FUNCTION "Indication" : Void   // FC11, SCL
{ S7_Optimized_Access := 'TRUE' }
VERSION : 0.1
BEGIN
   (*Управление индикацией*)
   //генератор импульсов
   "Timer_IND_1_DB".TON(IN := "Timer".IND_1_IN,
                        PT := "Timer".IND_1_PT,
                        Q => "Timer".IND_1_Q);
   "Timer_IND_2_DB".TON(IN := "Timer".IND_2_IN,
                        PT := "Timer".IND_2_PT,
                        Q => "Timer".IND_2_Q);
   "Timer".IND_1_PT := T#1s;
   "Timer".IND_2_PT := T#1s;
   IF NOT "Timer".IND_1_IN AND NOT "Timer".IND_2_IN THEN
       "Timer".IND_1_IN := TRUE;
   END_IF;
   IF "Timer".IND_1_Q THEN
       "Timer".IND_1_IN := FALSE;
       "Timer".IND_2_IN := TRUE;
       "Gen_imp" := FALSE;
   END_IF;
   IF "Timer".IND_2_Q THEN
       "Timer".IND_2_IN := FALSE;
       "Timer".IND_1_IN := TRUE;
       "Gen_imp" := TRUE;
   END_IF;

   (*Индикация «Работа»*)
   IF "Technology".Regim <> 5 AND
       "Technology".Regim <> 6 AND
       "Technology".Regim <> 7 AND
       "Technology".Regim <> 8 THEN
       "Sensors".Indication_RUN.Value := FALSE;
   END_IF;
   IF "Technology".Regim = 5 OR
       "Technology".Regim = 6 OR
       "Technology".Regim = 7 THEN
       "Sensors".Indication_RUN.Value := "Gen_imp";
   END_IF;
   IF "Technology".Regim = 8 THEN
       "Sensors".Indication_RUN.Value := TRUE;
   END_IF;

   (*Индикация «Авария»*)
   IF "Alarms_and_warnings".Alarm_P_gas_before_BG_max OR
       "Alarms_and_warnings".Alarm_P_gas_before_BG_min OR
       "Alarms_and_warnings".Alarm_P_gas_before_burner_min OR
       "Alarms_and_warnings".Alarm_P_gas_before_burner_max OR
       "Alarms_and_warnings".Alarm_DS_off OR
       "Alarms_and_warnings".Alarm_DV_off OR
       "Alarms_and_warnings".Alarm_dP_furnace_boiler_min OR
       "Alarms_and_warnings".Alarm_P_air_before_burner_min OR
       "Alarms_and_warnings".Alarm_P_water_after_boiler_min OR
       "Alarms_and_warnings".Alarm_P_water_after_boiler_max OR
       "Alarms_and_warnings".Alarm_T_water_after_boiler_max OR
       "Alarms_and_warnings".Alarm_Q_water_boiler_min OR
       "Alarms_and_warnings".Alarm_Not_flame_burner OR
       "Alarms_and_warnings".Alarm_stop_HMI OR
       "Alarms_and_warnings".Alarm_stop_SCADA OR
       "Alarms_and_warnings".Alarm_CO2_porog2 OR
       "Alarms_and_warnings".Alarm_CH4 THEN
       "Sensors".Indication_ALARM.Value := TRUE;
   ELSE
       IF "TON_alarm_1_DB".IN OR
           "TON_alarm_2_DB".IN OR
           "TON_alarm_3_DB".IN OR
           "TON_alarm_4_DB".IN OR
           "TON_alarm_5_DB".IN OR
           "TON_alarm_6_DB".IN OR
           "TON_alarm_7_DB".IN OR
           "TON_alarm_8_DB".IN OR
           "TON_alarm_9_DB".IN OR
           "TON_alarm_10_DB".IN OR
           "TON_alarm_11_DB".IN OR
           "TON_alarm_12_DB".IN OR
           "TON_alarm_13_DB".IN OR
           "FRONT_Btn_Alarm_stop_HMI" OR
           "FRONT_Btn_Alarm_stop_SCADA" OR
           "TON_alarm_14_DB".IN OR
           "TON_alarm_15_DB".IN THEN
           "Sensors".Indication_ALARM.Value := "Gen_imp";
       ELSE
           "Sensors".Indication_ALARM.Value := FALSE;
       END_IF;
   END_IF;

   (*Индикация «Защиты в норме»*)
   IF "Protections".Global THEN
       "Sensors".Indication_NORMA.Value := FALSE;
   ELSE
       IF "Protections".BLOCK_P_gas_before_BG_max OR
           "Protections".BLOCK_P_gas_before_BG_min OR
           "Protections".BLOCK_P_gas_before_burner_min OR
           "Protections".BLOCK_P_gas_before_burner_max OR
           "Protections".BLOCK_DS_off OR
           "Protections".BLOCK_DV_off OR
           "Protections".BLOCK_dP_in_furnance_min OR
           "Protections".BLOCK_P_air_before_burner_min OR
           "Protections".BLOCK_P_water_after_boiler_min OR
           "Protections".BLOCK_P_water_after_boiler_max OR
           "Protections".BLOCK_T_water_after_boiler_max OR
           "Protections".BLOCK_Q_water_boiler_min OR
           "Protections".BLOCK_Not_flame_burner OR
           "Protections".BLOCK_Alarm_stop_HMI OR
           "Protections".BLOCK_Alarm_stop_SCADA OR
           "Protections".BLOCK_CO2_porog2 OR
           "Protections".BLOCK_CH4 THEN
           "Sensors".Indication_NORMA.Value := "Gen_imp";
       ELSE
           "Sensors".Indication_NORMA.Value := TRUE;
       END_IF;
   END_IF;

   (*Индикация «Готов к розжигу»*)
   IF "Technology".Regim = 3 AND "Technology".Regim_ventilation_step = 25 THEN
       "Sensors".Indication_READY.Value := "Gen_imp";
   ELSE
       "Sensors".Indication_READY.Value := FALSE;
   END_IF;
END_FUNCTION

FUNCTION "Regim_map" : Void   // FC24, SCL
{ S7_Optimized_Access := 'TRUE' }
VERSION : 0.1
BEGIN
   (*Защита от неправильного ввода параметров режимной карты*)
   IF "RegMap".P_gaz_2 < "RegMap".P_gaz_1 THEN
       "RegMap".P_gaz_2 := "RegMap".P_gaz_1;
   END_IF;
   IF "RegMap".P_gaz_3 < "RegMap".P_gaz_2 THEN
       "RegMap".P_gaz_3 := "RegMap".P_gaz_2;
   END_IF;
   IF "RegMap".P_gaz_4 < "RegMap".P_gaz_3 THEN
       "RegMap".P_gaz_4 := "RegMap".P_gaz_3;
   END_IF;
   IF "RegMap".P_gaz_5 < "RegMap".P_gaz_4 THEN
       "RegMap".P_gaz_5 := "RegMap".P_gaz_4;
   END_IF;
   IF "RegMap".P_gaz_6 < "RegMap".P_gaz_5 THEN
       "RegMap".P_gaz_6 := "RegMap".P_gaz_5;
   END_IF;
   IF "RegMap".P_gaz_7 < "RegMap".P_gaz_6 THEN
       "RegMap".P_gaz_7 := "RegMap".P_gaz_6;
   END_IF;
   IF "RegMap".P_gaz_8 < "RegMap".P_gaz_7 THEN
       "RegMap".P_gaz_8 := "RegMap".P_gaz_7;
   END_IF;

   (*НАСТРОЙКА РЕЖИМНОЙ КАРТЫ*)
   (*давление воздуха*)
   "Polyline_P_air_DB"();

   "Polyline_P_air_DB".Input := "Sensors".P_gas_before_burner.Value;

   "Polyline_P_air_DB".UserData.Point[1].x := "RegMap".P_gaz_1;
   "Polyline_P_air_DB".UserData.Point[2].x := "RegMap".P_gaz_2;
   "Polyline_P_air_DB".UserData.Point[3].x := "RegMap".P_gaz_3;
   "Polyline_P_air_DB".UserData.Point[4].x := "RegMap".P_gaz_4;
   "Polyline_P_air_DB".UserData.Point[5].x := "RegMap".P_gaz_5;
   "Polyline_P_air_DB".UserData.Point[6].x := "RegMap".P_gaz_6;
   "Polyline_P_air_DB".UserData.Point[7].x := "RegMap".P_gaz_7;
   "Polyline_P_air_DB".UserData.Point[8].x := "RegMap".P_gaz_8;

   "Polyline_P_air_DB".UserData.Point[1].y := "RegMap".P_air_1;
   "Polyline_P_air_DB".UserData.Point[2].y := "RegMap".P_air_2;
   "Polyline_P_air_DB".UserData.Point[3].y := "RegMap".P_air_3;
   "Polyline_P_air_DB".UserData.Point[4].y := "RegMap".P_air_4;
   "Polyline_P_air_DB".UserData.Point[5].y := "RegMap".P_air_5;
   "Polyline_P_air_DB".UserData.Point[6].y := "RegMap".P_air_6;
   "Polyline_P_air_DB".UserData.Point[7].y := "RegMap".P_air_7;
   "Polyline_P_air_DB".UserData.Point[8].y := "RegMap".P_air_8;

   (*разряжение*)
   "Polyline_dP_DB"();

   "Polyline_dP_DB".Input := "Sensors".P_gas_before_burner.Value;

   "Polyline_dP_DB".UserData.Point[1].x := "RegMap".P_gaz_1;
   "Polyline_dP_DB".UserData.Point[2].x := "RegMap".P_gaz_2;
   "Polyline_dP_DB".UserData.Point[3].x := "RegMap".P_gaz_3;
   "Polyline_dP_DB".UserData.Point[4].x := "RegMap".P_gaz_4;
   "Polyline_dP_DB".UserData.Point[5].x := "RegMap".P_gaz_5;
   "Polyline_dP_DB".UserData.Point[6].x := "RegMap".P_gaz_6;
   "Polyline_dP_DB".UserData.Point[7].x := "RegMap".P_gaz_7;
   "Polyline_dP_DB".UserData.Point[8].x := "RegMap".P_gaz_8;

   "Polyline_dP_DB".UserData.Point[1].y := "RegMap".dP_furnace_1;
   "Polyline_dP_DB".UserData.Point[2].y := "RegMap".dP_furnace_2;
   "Polyline_dP_DB".UserData.Point[3].y := "RegMap".dP_furnace_3;
   "Polyline_dP_DB".UserData.Point[4].y := "RegMap".dP_furnace_4;
   "Polyline_dP_DB".UserData.Point[5].y := "RegMap".dP_furnace_5;
   "Polyline_dP_DB".UserData.Point[6].y := "RegMap".dP_furnace_6;
   "Polyline_dP_DB".UserData.Point[7].y := "RegMap".dP_furnace_7;
   "Polyline_dP_DB".UserData.Point[8].y := "RegMap".dP_furnace_8;

   (*Режимная карта. Применить. Для журнала событий*)
   IF "RegMap".Apply THEN
       "HMI".RegMap_Apply_Log := TRUE;
   END_IF;

   IF "Syst".First_scan_reg_map THEN
       "RegMap".Apply := TRUE;
       "Syst".First_scan_reg_map := FALSE;
   END_IF;

   //применить новые значения
   "Polyline_P_air_DB".Validate := "RegMap".Apply;
   "Polyline_dP_DB".Validate := "RegMap".Apply;
   IF "RegMap".Apply THEN
       "RegMap".Apply := FALSE;
   END_IF;

   //значение расчетных параметров
   "RegMap".P_air_regim_map := "Polyline_P_air_DB".Output;
   "RegMap".dP_furnace_regim_map := "Polyline_dP_DB".Output;

   //индикация ошибки
   "RegMap".Error := "Polyline_P_air_DB".Error OR "Polyline_dP_DB".Error;

   //сброс
   "Polyline_P_air_DB".Reset := "RegMap".Reset;
   "Polyline_dP_DB".Reset := "RegMap".Reset;
   IF "RegMap".Reset THEN
       "RegMap".Reset := FALSE;
   END_IF;
END_FUNCTION

FUNCTION "Control_Device" : Void   // FC25, SCL
{ S7_Optimized_Access := 'TRUE' }
VERSION : 0.1
BEGIN
   (*ДС. Ручное управление. Пуск. Для журнала событий*)
   IF "Control_DS".Manual_Start THEN
       "HMI".DS_Manual_Start_Log := TRUE;
   END_IF;
   (*ДС. Ручное управление. Стоп. Для журнала событий*)
   IF "Control_DS".Manual_Stop THEN
       "HMI".DS_Manual_Stop_Log := TRUE;
   END_IF;
   (*ДВ. Ручное управление. Пуск. Для журнала событий*)
   IF "Control_DV".Manual_Start THEN
       "HMI".DV_Manual_Start_Log := TRUE;
   END_IF;
   (*ДВ. Ручное управление. Стоп. Для журнала событий*)
   IF "Control_DV".Manual_Stop THEN
       "HMI".DV_Manual_Stop_Log := TRUE;
   END_IF;
   (*ЗДГ. Ручное управление. Открыть. Для журнала событий*)
   IF "Control_ZDG".Manual_open THEN
       "HMI".ZDG_Manual_open_Log := TRUE;
   END_IF;
   (*ЗДГ. Ручное управление. Закрыть. Для журнала событий*)
   IF "Control_ZDG".Manual_close THEN
       "HMI".ZDG_Manual_close_Log := TRUE;
   END_IF;
   (*ЗДГ. Ручное управление. Стоп. Для журнала событий*)
   IF "Control_ZDG".Manual_stop THEN
       "HMI".ZDG_Manual_stop_Log := TRUE;
   END_IF;
   (*ЗДСВ после котла. Ручное управление. Открыть. Для журнала событий*)
   IF "Control_ZDSV_after_boiler".Manual_open THEN
       "HMI".ZDSV_after_boiler_Manual_open_Log := TRUE;
   END_IF;
   (*ЗДСВ после котла. Ручное управление. Закрыть. Для журнала событий*)
   IF "Control_ZDSV_after_boiler".Manual_close THEN
       "HMI".ZDSV_after_boiler_Manual_close_Log := TRUE;
   END_IF;
   (*ЗДСВ после котла. Ручное управление. Стоп. Для журнала событий*)
   IF "Control_ZDSV_after_boiler".Manual_stop THEN
       "HMI".ZDSV_after_boiler_Manual_stop_Log := TRUE;
   END_IF;
   (*ЗДСВ перед котлом. Ручное управление. Открыть. Для журнала событий*)
   IF "Control_ZDSV_before_boiler".Manual_open THEN
       "HMI".ZDSV_before_boiler_Manual_open_Log := TRUE;
   END_IF;
   (*ЗДСВ перед котлом. Ручное управление. Закрыть. Для журнала событий*)
   IF "Control_ZDSV_before_boiler".Manual_close THEN
       "HMI".ZDSV_before_boiler_Manual_close_Log := TRUE;
   END_IF;
   (*ЗДСВ перед котлом. Ручное управление. Стоп. Для журнала событий*)
   IF "Control_ZDSV_before_boiler".Manual_stop THEN
       "HMI".ZDSV_before_boiler_Manual_stop_Log := TRUE;
   END_IF;

   (*Управление исполнительными механизмами*)
   (*ЗРГ*)
   //проверка и сброс ручных команд
   //сброс обеих команд при автоматическом режиме
   IF "Control_ZRG".Mode THEN
       "Control_ZRG".Manual_open := FALSE;
       "Control_ZRG".Manual_close := FALSE;
   END_IF;
   //сброс обеих команд при их одновременном наличии
   IF "Control_ZRG".Manual_open AND "Control_ZRG".Manual_close THEN
       "Control_ZRG".Manual_open := FALSE;
       "Control_ZRG".Manual_close := FALSE;
   END_IF;
   //сброс ручной команды на открытие при полном открытии
   IF "Sensors".ZRG_open.Value THEN
       "Control_ZRG".Manual_open := FALSE;
   END_IF;
   //сброс ручной команды на закрытие при полном закрытии
   IF "Sensors".ZRG_close.Value THEN
       "Control_ZRG".Manual_close := FALSE;
   END_IF;
   //проверка и сброс ручных команд от ПЛК
   //сброс обеих команд при режиме полного автомата
   IF "Control_ZRG".Mode_from_PLC THEN
       "Control_ZRG".Manual_open_from_PLC := FALSE;
       "Control_ZRG".Manual_close_from_PLC := FALSE;
   END_IF;
   //сброс обеих команд от ПЛК при их одновременном наличии
   IF "Control_ZRG".Manual_open_from_PLC AND "Control_ZRG".Manual_close_from_PLC THEN
       "Control_ZRG".Manual_open_from_PLC := FALSE;
       "Control_ZRG".Manual_close_from_PLC := FALSE;
   END_IF;
   //сброс ручной команды на открытие от ПЛК при полном открытии
   IF "Sensors".ZRG_open.Value THEN
       "Control_ZRG".Manual_open_from_PLC := FALSE;
   END_IF;
   //сброс ручной команды на закрытие от ПЛК при полном закрытии
   IF "Sensors".ZRG_close.Value THEN
       "Control_ZRG".Manual_close_from_PLC := FALSE;
   END_IF;
   //управление
   IF "Sensors".ZRG_avto.Value THEN
       IF "Technology".Regim <> 11 THEN
           "Control_ZRG".SP_PID := "Technology".SP_T_water_after_boiler;
       END_IF;
       "PID_impulse_ZRG_DB"(DIR := TRUE,
                            PV := "Sensors".T_water_after_boiler.Value,
                            SP := "Control_ZRG".SP_PID,
                            DB := "Control_ZRG".DB_PID,
                            KP := "Control_ZRG".KP_PID,
                            TI := "Control_ZRG".TI_PID,
                            TD := "Control_ZRG".TD_PID,
                            CYCLE := 100,
                            FMT := "Control_ZRG".FMT_PID,
                            DT_MIN := "Control_ZRG".DT_MIN_PID,
                            AUTO := ("Control_ZRG".Mode AND "Control_ZRG".Mode_from_PLC),
                            MORE := ((NOT "Control_ZRG".Mode AND "Control_ZRG".Manual_open) OR ("Control_ZRG".Mode AND "Control_ZRG".Manual_open_from_PLC)),
                            LESS := ((NOT "Control_ZRG".Mode AND "Control_ZRG".Manual_close) OR ("Control_ZRG".Mode AND "Control_ZRG".Manual_close_from_PLC)),
                            Hold := false,
                            GAP := "Control_ZRG".GAP,
                            PLUS := "Sensors".ZRG_control_open.Value,
                            MINUS := "Sensors".ZRG_control_close.Value);
   ELSE
       //при переводе БРУ в ручной режим
       "Sensors".ZRG_control_open.Value := FALSE;
       "Sensors".ZRG_control_close.Value := FALSE;
       "Control_ZRG".Manual_open := FALSE;
       "Control_ZRG".Manual_close := FALSE;
   END_IF;
   //ораничение на открытие по max давлению газа в режиме ПРОГРЕВ
   IF "Technology".Regim = 7 AND "Sensors".P_gas_before_burner.Value > "Technology".Max_P_gas_heating THEN
       "Sensors".ZRG_control_open.Value := FALSE;
   END_IF;
   //ограничение по закрытию ниже режима min мощности в режиме ПРОГРЕВ и РАБОТА
   IF ("Technology".Regim = 7 OR "Technology".Regim = 8) AND NOT "Sensors".ZRG_middle.Value THEN
       "Sensors".ZRG_control_close.Value := FALSE;
   END_IF;

   (*НАВ*)
   //проверка и сброс ручных команд
   //сброс обеих команд при автоматическом режиме
   IF "Control_NAV".Mode THEN
       "Control_NAV".Manual_open := FALSE;
       "Control_NAV".Manual_close := FALSE;
   END_IF;
   //сброс обеих команд при их одновременном наличии
   IF "Control_NAV".Manual_open AND "Control_NAV".Manual_close THEN
       "Control_NAV".Manual_open := FALSE;
       "Control_NAV".Manual_close := FALSE;
   END_IF;
   //сброс ручной команды на открытие при полном открытии
   IF "Sensors".NAV_open.Value THEN
       "Control_NAV".Manual_open := FALSE;
   END_IF;
   //сброс ручной команды на закрытие при полном закрытии
   IF "Sensors".NAV_close.Value THEN
       "Control_NAV".Manual_close := FALSE;
   END_IF;
   //проверка и сброс ручных команд от ПЛК
   //сброс обеих команд при режиме полного автомата
   IF "Control_NAV".Mode AND "Control_NAV".Mode_from_PLC THEN
       "Control_NAV".Manual_open_from_PLC := FALSE;
       "Control_NAV".Manual_close_from_PLC := FALSE;
   END_IF;
   //сброс обеих команд от ПЛК при их одновременном наличии
   IF "Control_NAV".Manual_open_from_PLC AND "Control_NAV".Manual_close_from_PLC THEN
       "Control_NAV".Manual_open_from_PLC := FALSE;
       "Control_NAV".Manual_close_from_PLC := FALSE;
   END_IF;
   //сброс ручной команды на открытие от ПЛК при полном открытии
   IF "Sensors".NAV_open.Value THEN
       "Control_NAV".Manual_open_from_PLC := FALSE;
   END_IF;
   //сброс ручной команды на закрытие от ПЛК при полном закрытии
   IF "Sensors".NAV_close.Value THEN
       "Control_NAV".Manual_close_from_PLC := FALSE;
   END_IF;
   //управление
   IF "Sensors".NAV_avto.Value THEN
       "PID_impulse_NAV_DB"(DIR := TRUE,
                            PV := "Sensors".P_air_burner.Value,
                            SP := "Control_NAV".SP_PID,
                            DB := "Control_NAV".DB_PID,
                            KP := "Control_NAV".KP_PID,
                            TI := "Control_NAV".TI_PID,
                            TD := "Control_NAV".TD_PID,
                            CYCLE := 100,
                            FMT := "Control_NAV".FMT_PID,
                            DT_MIN := "Control_NAV".DT_MIN_PID,
                            AUTO := ("Control_NAV".Mode AND "Control_NAV".Mode_from_PLC),
                            MORE := ((NOT "Control_NAV".Mode AND "Control_NAV".Manual_open) OR ("Control_NAV".Mode AND "Control_NAV".Manual_open_from_PLC)),
                            LESS := ((NOT "Control_NAV".Mode AND "Control_NAV".Manual_close) OR ("Control_NAV".Mode AND "Control_NAV".Manual_close_from_PLC)),
                            Hold := false,
                            GAP := "Control_NAV".GAP,
                            PLUS := "Sensors".NAV_control_open.Value,
                            MINUS := "Sensors".NAV_control_close.Value);
   ELSE
       //при переводе БРУ в ручной режим
       "Sensors".NAV_control_open.Value := FALSE;
       "Sensors".NAV_control_close.Value := FALSE;
       "Control_NAV".Manual_open := FALSE;
       "Control_NAV".Manual_close := FALSE;
   END_IF;

   (*НАД*)
   //проверка и сброс ручных команд
   //сброс обеих команд при автоматическом режиме
   IF "Control_NAD".Mode THEN
       "Control_NAD".Manual_open := FALSE;
       "Control_NAD".Manual_close := FALSE;
   END_IF;
   //сброс обеих команд при их одновременном наличии
   IF "Control_NAD".Manual_open AND "Control_NAD".Manual_close THEN
       "Control_NAD".Manual_open := FALSE;
       "Control_NAD".Manual_close := FALSE;
   END_IF;
   //сброс ручной команды на открытие при полном открытии
   IF "Sensors".NAD_open.Value THEN
       "Control_NAD".Manual_open := FALSE;
   END_IF;
   //сброс ручной команды на закрытие при полном закрытии
   IF "Sensors".NAD_close.Value THEN
       "Control_NAD".Manual_close := FALSE;
   END_IF;
   //проверка и сброс ручных команд от ПЛК
   //сброс обеих команд при режиме полного автомата
   IF "Control_NAD".Mode AND "Control_NAD".Mode_from_PLC THEN
       "Control_NAD".Manual_open_from_PLC := FALSE;
       "Control_NAD".Manual_close_from_PLC := FALSE;
   END_IF;
   //сброс обеих команд от ПЛК при их одновременном наличии
   IF "Control_NAD".Manual_open_from_PLC AND "Control_NAD".Manual_close_from_PLC THEN
       "Control_NAD".Manual_open_from_PLC := FALSE;
       "Control_NAD".Manual_close_from_PLC := FALSE;
   END_IF;
   //сброс ручной команды на открытие от ПЛК при полном открытии
   IF "Sensors".NAD_open.Value THEN
       "Control_NAD".Manual_open_from_PLC := FALSE;
   END_IF;
   //сброс ручной команды на закрытие от ПЛК при полном закрытии
   IF "Sensors".NAD_close.Value THEN
       "Control_NAD".Manual_close_from_PLC := FALSE;
   END_IF;
   //управление
   IF "Sensors".NAD_avto.Value THEN
       "PID_impulse_NAD_DB"(DIR := FALSE,
                            PV := "Sensors".dP_furnace_boiler.Value,
                            SP := "Control_NAD".SP_PID,
                            DB := "Control_NAD".DB_PID,
                            KP := "Control_NAD".KP_PID,
                            TI := "Control_NAD".TI_PID,
                            TD := "Control_NAD".TD_PID,
                            CYCLE := 100,
                            FMT := "Control_NAD".FMT_PID,
                            DT_MIN := "Control_NAD".DT_MIN_PID,
                            AUTO := ("Control_NAD".Mode AND "Control_NAD".Mode_from_PLC),
                            MORE := ((NOT "Control_NAD".Mode AND "Control_NAD".Manual_open) OR ("Control_NAD".Mode AND "Control_NAD".Manual_open_from_PLC)),
                            LESS := ((NOT "Control_NAD".Mode AND "Control_NAD".Manual_close) OR ("Control_NAD".Mode AND "Control_NAD".Manual_close_from_PLC)),
                            Hold := false,
                            GAP := "Control_NAD".GAP,
                            PLUS := "Sensors".NAD_control_open.Value,
                            MINUS := "Sensors".NAD_control_close.Value);
   ELSE
       //при переводе БРУ в ручной режим
       "Sensors".NAD_control_open.Value := FALSE;
       "Sensors".NAD_control_close.Value := FALSE;
       "Control_NAD".Manual_open := FALSE;
       "Control_NAD".Manual_close := FALSE;
   END_IF;

   (*ЗДГ*)
   //Проверка и сброс ручных команд
   //Сброс всех команд при автоматическом режиме
   IF "Control_ZDG".Mode THEN
       "Control_ZDG".Manual_open := FALSE;
       "Control_ZDG".Manual_close := FALSE;
       "Control_ZDG".Manual_stop := FALSE;
   END_IF;
   //сброс обеих команд при их одновременном наличии
   IF "Control_ZDG".Manual_open AND "Control_ZDG".Manual_close THEN
       "Control_ZDG".Manual_open := FALSE;
       "Control_ZDG".Manual_close := FALSE;
   END_IF;
   //сброс ручных команд при начале движения
   IF "Sensors".ZDG_opening.Value OR "Sensors".ZDG_closing.Value THEN
       "Control_ZDG".Manual_open := FALSE;
       "Control_ZDG".Manual_close := FALSE;
   END_IF;
   //сброс команды стоп при окончаниии движения
   IF NOT "Sensors".ZDG_opening.Value AND NOT "Sensors".ZDG_closing.Value THEN
       "Control_ZDG".Manual_stop := FALSE;
   END_IF;
   //сброс команды открыть при полном открытии или запрете
   IF NOT "Sensors".ZDG_no_open.Value OR "Sensors".ZDG_control_disable_open.Value THEN
       "Control_ZDG".Manual_open := FALSE;
   END_IF;
   //сброс команды закрыть при полном закрытии
   IF NOT "Sensors".ZDG_no_close.Value THEN
       "Control_ZDG".Manual_close := FALSE;
   END_IF;
   //Проверка и сброс автоматических команд
   //сброс обеих команд при их одновременном наличии
   IF "Control_ZDG".Avto_open AND "Control_ZDG".Avto_close THEN
       "Control_ZDG".Avto_open := FALSE;
       "Control_ZDG".Avto_close := FALSE;
   END_IF;
   //сброс команд при начале движения
   IF "Sensors".ZDG_opening.Value OR "Sensors".ZDG_closing.Value THEN
       "Control_ZDG".Avto_open := FALSE;
       "Control_ZDG".Avto_close := FALSE;
   END_IF;
   //сброс команды стоп при окончаниии движения
   IF NOT "Sensors".ZDG_opening.Value AND NOT "Sensors".ZDG_closing.Value THEN
       "Control_ZDG".Avto_stop := FALSE;
   END_IF;
   //сброс команды открыть при полном открытии или запрете
   IF NOT "Sensors".ZDG_no_open.Value OR "Sensors".ZDG_control_disable_open.Value THEN
       "Control_ZDG".Avto_open := FALSE;
   END_IF;
   //сброс команды закрыть при полном закрытии
   IF NOT "Sensors".ZDG_no_close.Value THEN
       "Control_ZDG".Avto_close := FALSE;
   END_IF;
   //управление
   IF "Control_ZDG".Mode THEN
       // автоматический режим
       "Sensors".ZDG_control_open.Value := "Control_ZDG".Avto_open;
       "Sensors".ZDG_control_close.Value := "Control_ZDG".Avto_close;
       "Sensors".ZDG_control_stop.Value := "Control_ZDG".Avto_stop;
   ELSE
       //ручной режим
       "Sensors".ZDG_control_open.Value := "Control_ZDG".Manual_open;
       "Sensors".ZDG_control_close.Value := "Control_ZDG".Manual_close;
       "Sensors".ZDG_control_stop.Value := "Control_ZDG".Manual_stop;
   END_IF;
   //Управление запретом открытия
   IF "Sensors".PZK1_open.Value OR                                          //ПЗК1 открыт
       ("Sensors".PZK2_open.Value OR "Sensors".PZK2_not_close.Value) OR     //ПЗК2 открыт
       ("Sensors".Q_water_boiler_min.Value AND NOT "Protections".BLOCK_Q_water_boiler_min) OR    //нет расхода воды
       (NOT "Sensors".DV_invertor_on.Value AND NOT "Sensors".DV_powergrid_on.Value) THEN //ДВ  
       "Sensors".ZDG_control_disable_open.Value := TRUE;
   ELSE
       "Sensors".ZDG_control_disable_open.Value := FALSE;
   END_IF;

   (*КБ*)
   //при переходе из автоматического в ручной режим управления в ручную команду копируем текущее положение
   "F_TRIG_KB_DB"(CLK := "Control_KB".Mode,
                  Q => "FRONT_KB_mode");
   IF "FRONT_KB_mode" THEN
       "Control_KB".Manual_close := "Sensors".KB_close.Value;
   END_IF;
   //управление
   IF "Control_KB".Mode THEN
       // автоматический режим
       "Sensors".KB_control_close.Value := "Control_KB".Avto_close;
   ELSE
       //ручной режим
       "Sensors".KB_control_close.Value := "Control_KB".Manual_close;
   END_IF;

   (*КО*)
   //при переходе из автоматического в ручной режим управления в ручную команду копируем текущее положение
   "F_TRIG_KO_DB"(CLK := "Control_KO".Mode,
                  Q => "FRONT_KO_mode");
   IF "FRONT_KO_mode" THEN
       "Control_KO".Manual_open := "Sensors".KO_open.Value;
   END_IF;
   //управление
   IF "Control_KO".Mode THEN
       // автоматический режим
       "Sensors".KO_control_open.Value := "Control_KO".Avto_open;
   ELSE
       //ручной режим
       "Sensors".KO_control_open.Value := "Control_KO".Manual_open;
   END_IF;

   (*КЗ*)
   //при переходе из автоматического в ручной режим управления в ручную команду копируем текущее положение
   "F_TRIG_KZ_DB"(CLK := "Control_KZ".Mode,
                  Q => "FRONT_KZ_mode");
   IF "FRONT_KZ_mode" THEN
       "Control_KZ".Manual_open := "Sensors".KZ_open.Value;
   END_IF;
   //закрытие клапана запальника по таймеру
   "TON_close_KZ_DB".TON(IN := "Timer".close_KZ_IN,
                         PT := T#25s,
                         Q => "Timer".close_KZ_Q);
   IF "Timer".close_KZ_Q THEN
       "Timer".close_KZ_IN := FALSE;
       "Control_KZ".Avto_open := FALSE;
   END_IF;
   //управление
   IF "Control_KZ".Mode THEN
       // автоматический режим
       "Sensors".KZ_control_open.Value := "Control_KZ".Avto_open;
   ELSE
       //ручной режим
       "Sensors".KZ_control_open.Value := "Control_KZ".Manual_open;
   END_IF;

   (*ИВН*)
   //при переходе из автоматического в ручной режим управления в ручную команду копируем текущую команду
   "F_TRIG_IVN_DB"(CLK := "Control_IVN".Mode,
                   Q => "FRONT_IVN_mode");
   IF "FRONT_IVN_mode" THEN
       "Control_IVN".Manual_on := "Control_IVN".Avto_on;
   END_IF;
   //сброс автоматической команды на включения через 6 секунд
   "TON_avto_reset_IVN_DB".TON(IN := "Sensors".IVN_control_on.Value,
                               PT := T#6s,
                               Q => "Timer".avto_reset_IVN_Q);
   IF "Timer".avto_reset_IVN_Q THEN
       "Control_IVN".Avto_on := FALSE;
   END_IF;
   //управление
   IF "Control_IVN".Mode THEN
       // автоматический режим
       "Sensors".IVN_control_on.Value := "Control_IVN".Avto_on;
   ELSE
       //ручной режим
       "Sensors".IVN_control_on.Value := "Control_IVN".Manual_on;
   END_IF;

   (*ПЗК1*)
   //при переходе из автоматического в ручной режим управления в ручную команду копируем текущее положение
   "F_TRIG_PZK1_DB"(CLK := "Control_PZK1".Mode,
                    Q => "FRONT_PZK1_mode");
   IF "FRONT_PZK1_mode" THEN
       "Control_PZK1".Manual_open := "Sensors".PZK1_open.Value;
   END_IF;
   IF "Control_PZK1".Mode THEN
       // автоматический режим
       "Sensors".PZK1_control_open.Value := "Control_PZK1".Avto_open;
   ELSE
       //ручной режим
       "Sensors".PZK1_control_open.Value := "Control_PZK1".Manual_open;
   END_IF;

   (*ПЗК2*)
   //при переходе из автоматического в ручной режим управления в ручную команду копируем текущее положение
   "F_TRIG_PZK2_DB"(CLK := "Control_PZK2".Mode,
                    Q => "FRONT_PZK2_mode");
   IF "FRONT_PZK2_mode" THEN
       "Control_PZK2".Manual_open := "Sensors".PZK2_open.Value;
   END_IF;
   IF "Control_PZK2".Mode THEN
       // автоматический режим
       "Sensors".PZK2_control_open.Value := "Control_PZK2".Avto_open;
   ELSE
       //ручной режим
       "Sensors".PZK2_control_open.Value := "Control_PZK2".Manual_open;
   END_IF;

   (*ЗДСВ перед котлом*)
   //Проверка и сброс ручных команд
   //Сброс всех команд при автоматическом режиме
   IF "Control_ZDSV_before_boiler".Mode THEN
       "Control_ZDSV_before_boiler".Manual_open := FALSE;
       "Control_ZDSV_before_boiler".Manual_close := FALSE;
       "Control_ZDSV_before_boiler".Manual_stop := FALSE;
   END_IF;
   //сброс обеих команд при их одновременном наличии
   IF "Control_ZDSV_before_boiler".Manual_open AND "Control_ZDSV_before_boiler".Manual_close THEN
       "Control_ZDSV_before_boiler".Manual_open := FALSE;
       "Control_ZDSV_before_boiler".Manual_close := FALSE;
   END_IF;
   //сброс ручных команд при начале движения
   IF "Sensors".ZDSV_before_boiler_opening.Value OR "Sensors".ZDSV_before_boiler_closing.Value THEN
       "Control_ZDSV_before_boiler".Manual_open := FALSE;
       "Control_ZDSV_before_boiler".Manual_close := FALSE;
   END_IF;
   //сброс команды стоп при окончаниии движения
   IF NOT "Sensors".ZDSV_before_boiler_opening.Value AND NOT "Sensors".ZDSV_before_boiler_closing.Value THEN
       "Control_ZDSV_before_boiler".Manual_stop := FALSE;
   END_IF;
   //сброс команды открыть при полном открытии
   IF NOT "Sensors".ZDSV_before_boiler_no_open.Value THEN
       "Control_ZDSV_before_boiler".Manual_open := FALSE;
   END_IF;
   //сброс команды закрыть при полном закрытии или запрете
   IF NOT "Sensors".ZDSV_before_boiler_no_close.Value OR "Sensors".ZDSV_before_boiler_control_disable_close.Value THEN
       "Control_ZDSV_before_boiler".Manual_close := FALSE;
   END_IF;
   //Проверка и сброс автоматических команд
   //сброс обеих команд при их одновременном наличии
   IF "Control_ZDSV_before_boiler".Avto_open AND "Control_ZDSV_before_boiler".Avto_close THEN
       "Control_ZDSV_before_boiler".Avto_open := FALSE;
       "Control_ZDSV_before_boiler".Avto_close := FALSE;
   END_IF;
   //сброс ручных команд при начале движения
   IF "Sensors".ZDSV_before_boiler_opening.Value OR "Sensors".ZDSV_before_boiler_closing.Value THEN
       "Control_ZDSV_before_boiler".Avto_open := FALSE;
       "Control_ZDSV_before_boiler".Avto_close := FALSE;
   END_IF;
   //сброс команды стоп при окончаниии движения
   IF NOT "Sensors".ZDSV_before_boiler_opening.Value AND NOT "Sensors".ZDSV_before_boiler_closing.Value THEN
       "Control_ZDSV_before_boiler".Avto_stop := FALSE;
   END_IF;
   //сброс команды открыть при полном открытии
   IF NOT "Sensors".ZDSV_before_boiler_no_open.Value THEN
       "Control_ZDSV_before_boiler".Avto_open := FALSE;
   END_IF;
   //сброс команды закрыть при полном закрытии или запрете
   IF NOT "Sensors".ZDSV_before_boiler_no_close.Value OR "Sensors".ZDSV_before_boiler_control_disable_close.Value THEN
       "Control_ZDSV_before_boiler".Avto_close := FALSE;
   END_IF;
   //управление
   IF "Control_ZDSV_before_boiler".Mode THEN
       // автоматический режим
       "Sensors".ZDSV_before_boiler_control_open.Value := "Control_ZDSV_before_boiler".Avto_open;
       "Sensors".ZDSV_before_boiler_control_close.Value := "Control_ZDSV_before_boiler".Avto_close;
       "Sensors".ZDSV_before_boiler_control_stop.Value := "Control_ZDSV_before_boiler".Avto_stop;
   ELSE
       //ручной режим
       "Sensors".ZDSV_before_boiler_control_open.Value := "Control_ZDSV_before_boiler".Manual_open;
       "Sensors".ZDSV_before_boiler_control_close.Value := "Control_ZDSV_before_boiler".Manual_close;
       "Sensors".ZDSV_before_boiler_control_stop.Value := "Control_ZDSV_before_boiler".Manual_stop;
   END_IF;
   //Управление запретом закрытия
   IF "Sensors".ZDG_no_close.Value OR                              //ЗДГ не закрыта
       ("Sensors".T_water_after_boiler_max.Value AND NOT "Protections".BLOCK_T_water_after_boiler_max) THEN               //Перегрев котла
       "Sensors".ZDSV_before_boiler_control_disable_close.Value := TRUE;
   ELSE
       "Sensors".ZDSV_before_boiler_control_disable_close.Value := FALSE;
   END_IF;

   (*Задвижка сетевой воды после котла*)
   //Проверка и сброс ручных команд
   //Сброс всех команд при автоматическом режиме
   IF "Control_ZDSV_after_boiler".Mode THEN
       "Control_ZDSV_after_boiler".Manual_open := FALSE;
       "Control_ZDSV_after_boiler".Manual_close := FALSE;
       "Control_ZDSV_after_boiler".Manual_stop := FALSE;
   END_IF;
   //сброс обоих команд при их одновременном наличии
   IF "Control_ZDSV_after_boiler".Manual_open AND "Control_ZDSV_after_boiler".Manual_close THEN
       "Control_ZDSV_after_boiler".Manual_open := FALSE;
       "Control_ZDSV_after_boiler".Manual_close := FALSE;
   END_IF;
   //сброс ручных команд при начале движения
   IF "Sensors".ZDSV_after_boiler_opening.Value OR "Sensors".ZDSV_after_boiler_closing.Value THEN
       "Control_ZDSV_after_boiler".Manual_open := FALSE;
       "Control_ZDSV_after_boiler".Manual_close := FALSE;
   END_IF;
   //сброс команды стоп при окончаниии движения
   IF NOT "Sensors".ZDSV_after_boiler_opening.Value AND NOT "Sensors".ZDSV_after_boiler_closing.Value THEN
       "Control_ZDSV_after_boiler".Manual_stop := FALSE;
   END_IF;
   //сброс команды открыть при полном открытии
   IF NOT "Sensors".ZDSV_after_boiler_no_open.Value THEN
       "Control_ZDSV_after_boiler".Manual_open := FALSE;
   END_IF;
   //сброс команды закрыть при полном закрытии или запрете
   IF NOT "Sensors".ZDSV_after_boiler_no_close.Value OR "Sensors".ZDSV_after_boiler_control_disable_close.Value THEN
       "Control_ZDSV_after_boiler".Manual_close := FALSE;
   END_IF;
   //Проверка и сброс автоматических команд
   //сброс обоих команд при их одновременном наличии
   IF "Control_ZDSV_after_boiler".Avto_open AND "Control_ZDSV_after_boiler".Avto_close THEN
       "Control_ZDSV_after_boiler".Avto_open := FALSE;
       "Control_ZDSV_after_boiler".Avto_close := FALSE;
   END_IF;
   //сброс ручных команд при начале движения
   IF "Sensors".ZDSV_after_boiler_opening.Value OR "Sensors".ZDSV_after_boiler_closing.Value THEN
       "Control_ZDSV_after_boiler".Avto_open := FALSE;
       "Control_ZDSV_after_boiler".Avto_close := FALSE;
   END_IF;
   //сброс команды стоп при окончаниии движения
   IF NOT "Sensors".ZDSV_after_boiler_opening.Value AND NOT "Sensors".ZDSV_after_boiler_closing.Value THEN
       "Control_ZDSV_after_boiler".Avto_stop := FALSE;
   END_IF;
   //сброс команды открыть при полном открытии
   IF NOT "Sensors".ZDSV_after_boiler_no_open.Value THEN
       "Control_ZDSV_after_boiler".Avto_open := FALSE;
   END_IF;
   //сброс команды закрыть при полном закрытии или запрете
   IF NOT "Sensors".ZDSV_after_boiler_no_close.Value OR "Sensors".ZDSV_after_boiler_control_disable_close.Value THEN
       "Control_ZDSV_after_boiler".Avto_close := FALSE;
   END_IF;
   //управление
   IF "Control_ZDSV_after_boiler".Mode THEN
       // автоматический режим
       "Sensors".ZDSV_after_boiler_control_open.Value := "Control_ZDSV_after_boiler".Avto_open;
       "Sensors".ZDSV_after_boiler_control_close.Value := "Control_ZDSV_after_boiler".Avto_close;
       "Sensors".ZDSV_after_boiler_control_stop.Value := "Control_ZDSV_after_boiler".Avto_stop;
   ELSE
       //ручной режим
       "Sensors".ZDSV_after_boiler_control_open.Value := "Control_ZDSV_after_boiler".Manual_open;
       "Sensors".ZDSV_after_boiler_control_close.Value := "Control_ZDSV_after_boiler".Manual_close;
       "Sensors".ZDSV_after_boiler_control_stop.Value := "Control_ZDSV_after_boiler".Manual_stop;
   END_IF;
   //Управление запретом закрытия
   IF "Sensors".ZDSV_before_boiler_no_close.Value OR       //ЗДСВ перед котлом не закрыта
       (NOT "Sensors".P_water_after_boiler_min.Value AND NOT "Protections".BLOCK_P_water_after_boiler_min) OR     //P после котла больше min 
       ("Sensors".T_water_after_boiler_max.Value AND NOT "Protections".BLOCK_T_water_after_boiler_max) THEN       //Перегрев котла
       "Sensors".ZDSV_after_boiler_control_disable_close.Value := TRUE;
   ELSE
       "Sensors".ZDSV_after_boiler_control_disable_close.Value := FALSE;
   END_IF;

   (*ДВ*)
   //Проверка и сброс ручных команд
   //Сброс команд при автоматическом режиме
   IF "Control_DV".Mode THEN
       "Control_DV".Manual_Start := FALSE;
       "Control_DV".Manual_Stop := FALSE;
   END_IF;
   "F_TRIG_DV_DB"(CLK := "Control_DV".Mode,
                  Q => "FRONT_DV_mode");
   IF "FRONT_DV_mode" THEN
       "Control_DV".Manual_frequency := "PID_analog_DV_DB".OUT;
   END_IF;
   //обеих команд при их одновременном наличии или отсутствии дистанционного режима
   IF ("Control_DV".Manual_Start AND "Control_DV".Manual_Stop) OR
       NOT "Sensors".DV_dist_control.Value THEN
       "Control_DV".Manual_Start := FALSE;
       "Control_DV".Manual_Stop := FALSE;
   END_IF;
   //Подача команды на отключение при аварии ПЧ
   IF NOT "Control_DV".Mode AND "Alarms_and_warnings".Warning_DV_invertor_alarm AND "Sensors".DV_invertor_on.Value THEN
       "Control_DV".Manual_Stop := TRUE;
   END_IF;
   //сброс команды пуск после включения
   IF "Sensors".DV_invertor_on.Value OR "Sensors".DV_powergrid_on.Value THEN
       "Control_DV".Manual_Start := FALSE;
   END_IF;
   //сброс команды пуск и подача команды стоп при отключенном ДС
   (*IF NOT "Sensors".DS_invertor_on.Value AND NOT "Sensors".DS_powergrid_on.Value THEN
       "Control_DV".Manual_Start := FALSE;
   END_IF;*)
   //сброс команды стоп после отключения
   IF NOT "Sensors".DV_invertor_on.Value AND NOT "Sensors".DV_powergrid_on.Value THEN
       "Control_DV".Manual_Stop := FALSE;
   END_IF;
   //Проверка и сброс автоматических команд
   //сброс обеих команд при их одновременном наличии
   IF "Control_DV".Avto_Start AND "Control_DV".Avto_Stop THEN
       "Control_DV".Avto_Start := FALSE;
       "Control_DV".Avto_Stop := FALSE;
   END_IF;
   //Подача команды на отключение при аварии ПЧ
   IF "Control_DV".Mode AND "Alarms_and_warnings".Warning_DV_invertor_alarm AND "Sensors".DV_invertor_on.Value THEN
       "Control_DV".Avto_Stop := TRUE;
   END_IF;
   IF "Alarms_and_warnings".Warning_DV_invertor_alarm AND "Sensors".DV_invertor_mode.Value THEN
       "Control_DV".Avto_Start := FALSE;
   END_IF;
   //сброс команды пуск после включения
   IF "Sensors".DV_invertor_on.Value OR "Sensors".DV_powergrid_on.Value THEN
       "Control_DV".Avto_Start := FALSE;
   END_IF;
   //сброс команды стоп после отключения
   IF NOT "Sensors".DV_invertor_on.Value AND NOT "Sensors".DV_powergrid_on.Value THEN
       "Control_DV".Avto_Stop := FALSE;
   END_IF;
   //управление
   IF "Sensors".DV_dist_control.Value THEN    //Управление «Дистанционный» ДВ
       //включение
       IF "Control_DV".Mode THEN
           // автоматический режим
           "Sensors".DV_control_start.Value := "Control_DV".Avto_Start;
           "Sensors".DV_control_stop.Value := "Control_DV".Avto_Stop;
       ELSE
           //ручной режим
           "Sensors".DV_control_start.Value := "Control_DV".Manual_Start;
           "Sensors".DV_control_stop.Value := "Control_DV".Manual_Stop;
       END_IF;
       //частота
       IF "Sensors".DV_invertor_mode.Value THEN    //Режим "ПЧ" ДВ
           "PID_analog_DV_DB"(AUTO := ("Control_DV".Mode AND "Control_DV".Mode_from_PLC),
                              DIR := TRUE,
                              PV := "Sensors".P_air_burner.Value,
                              SP := "Control_DV".SP_PID,
                              DB := "Control_DV".DB_PID,
                              KP := "Control_DV".KP_PID,
                              TI := "Control_DV".TI_PID,
                              TD := "Control_DV".TD_PID,
                              CYCLE := 100,
                              Hold := false,
                              OUT_MIN := "Sensors".DV_control_frequency.Low_limit_phisical_current,
                              OUT_MAX := "Sensors".DV_control_frequency.High_limit_phisical_current,
                              OUT := "Sensors".DV_control_frequency.Value);
           IF "Control_DV".Mode THEN
               "PID_analog_DV_DB".OUT_MAN := "Control_DV".Manual_frequency_from_PLC;
           ELSE
               "PID_analog_DV_DB".OUT_MAN := "Control_DV".Manual_frequency;
           END_IF;
       ELSE
           //"PID_analog_DV_DB".Hold := TRUE;
           "Sensors".DV_control_frequency.Value := 0.0;
       END_IF;
   ELSE
       "Sensors".DV_control_start.Value := FALSE;
       "Sensors".DV_control_stop.Value := FALSE;
       "Sensors".DV_control_frequency.Value := 0.0;
   END_IF;

   (*ДС*)
   //Проверка и сброс ручных команд
   //Сброс команд при автоматическом режиме
   IF "Control_DS".Mode THEN
       "Control_DS".Manual_Start := FALSE;
       "Control_DS".Manual_Stop := FALSE;
   END_IF;
   "F_TRIG_DS_DB"(CLK := "Control_DS".Mode,
                  Q => "FRONT_DS_mode");
   IF "FRONT_DS_mode" THEN
       "Control_DS".Manual_frequency := "PID_analog_DS_DB".OUT;
   END_IF;
   //сброс обоих команд при их одновременном наличии или отсутствии дистанционного режима
   IF ("Control_DS".Manual_Start AND "Control_DS".Manual_Stop) OR
       NOT "Sensors".DS_dist_control.Value THEN
       "Control_DS".Manual_Start := FALSE;
       "Control_DS".Manual_Stop := FALSE;
   END_IF;
   //Подача команды на отключение при аварии ПЧ
   IF NOT "Control_DS".Mode AND "Alarms_and_warnings".Warning_DS_invertor_alarm AND "Sensors".DS_invertor_on.Value THEN
       "Control_DS".Manual_Stop := TRUE;
   END_IF;
   //сброс команды пуск после включения
   IF "Sensors".DS_invertor_on.Value OR "Sensors".DS_powergrid_on.Value THEN
       "Control_DS".Manual_Start := FALSE;
   END_IF;
   //сброс команды стоп после отключения
   IF NOT "Sensors".DS_invertor_on.Value AND NOT "Sensors".DS_powergrid_on.Value THEN
       "Control_DS".Manual_Stop := FALSE;
   END_IF;
   //Проверка и сброс автоматических команд
   //сброс обоих команд при их одновременном наличии
   IF "Control_DS".Avto_Start AND "Control_DS".Avto_Stop THEN
       "Control_DS".Avto_Start := FALSE;
       "Control_DS".Avto_Stop := FALSE;
   END_IF;
   //Подача команды на отключение при аварии ПЧ
   IF "Control_DS".Mode AND "Alarms_and_warnings".Warning_DS_invertor_alarm AND "Sensors".DS_invertor_on.Value THEN
       "Control_DS".Avto_Stop := TRUE;
   END_IF;
   IF "Alarms_and_warnings".Warning_DS_invertor_alarm AND "Sensors".DS_invertor_mode.Value THEN
       "Control_DS".Avto_Start := FALSE;
   END_IF;
   //сброс команды пуск после включения
   IF "Sensors".DS_invertor_on.Value OR "Sensors".DS_powergrid_on.Value THEN
       "Control_DS".Avto_Start := FALSE;
   END_IF;
   //сброс команды стоп после отключения
   IF NOT "Sensors".DS_invertor_on.Value AND NOT "Sensors".DS_powergrid_on.Value THEN
       "Control_DS".Avto_Stop := FALSE;
   END_IF;
   //управление
   IF "Sensors".DS_dist_control.Value THEN    //Управление «Дистанционный» ДС
       //включение
       IF "Control_DS".Mode THEN
           // автоматический режим
           "Sensors".DS_control_start.Value := "Control_DS".Avto_Start;
           "Sensors".DS_control_stop.Value := "Control_DS".Avto_Stop;
       ELSE
           //ручной режим
           "Sensors".DS_control_start.Value := "Control_DS".Manual_Start;
           "Sensors".DS_control_stop.Value := "Control_DS".Manual_Stop;
       END_IF;
       //частота
       IF "Sensors".DS_invertor_mode.Value THEN    //Режим "ПЧ" ДС
           "PID_analog_DS_DB"(AUTO := ("Control_DS".Mode AND "Control_DS".Mode_from_PLC),
                              DIR := FALSE,
                              PV := "Sensors".dP_furnace_boiler.Value,
                              SP := "Control_DS".SP_PID,
                              DB := "Control_DS".DB_PID,
                              KP := "Control_DS".KP_PID,
                              TI := "Control_DS".TI_PID,
                              TD := "Control_DS".TD_PID,
                              CYCLE := 100,
                              Hold := false,
                              OUT_MIN := "Sensors".DS_control_frequency.Low_limit_phisical_current,
                              OUT_MAX := "Sensors".DS_control_frequency.High_limit_phisical_current,
                              OUT := "Sensors".DS_control_frequency.Value);
           IF "Control_DS".Mode THEN
               "PID_analog_DS_DB".OUT_MAN := "Control_DS".Manual_frequency_from_PLC;
           ELSE
               "PID_analog_DS_DB".OUT_MAN := "Control_DS".Manual_frequency;
           END_IF;
       ELSE
           //"PID_analog_DS_DB".Hold := TRUE;
           "Sensors".DS_control_frequency.Value := 0.0;
       END_IF;
   ELSE
       "Sensors".DS_control_start.Value := FALSE;
       "Sensors".DS_control_stop.Value := FALSE;
       "Sensors".DS_control_frequency.Value := 0.0;
   END_IF;
END_FUNCTION

FUNCTION "HMI_and_SCADA" : Void   // FC26, SCL
{ S7_Optimized_Access := 'TRUE' }
VERSION : 0.1
BEGIN
   //кнопка ВЕНТИЛЯЦИЯ на панели оператора
   "R_TRIG_DB"(CLK := "HMI".Btn_Ventilation_HMI,
               Q => "FRONT_Btn_Ventilation_HMI");
   IF "FRONT_Btn_Ventilation_HMI" THEN
       "HMI".Btn_Ventilation_HMI := FALSE;
   END_IF;
   //кнопка ВЕНТИЛЯЦИЯ на SCADA
   "R_TRIG_DB_1"(CLK := "HMI".Btn_Ventilation_SCADA,
                 Q => "FRONT_Btn_Ventilation_SCADA");
   IF "FRONT_Btn_Ventilation_SCADA" THEN
       "HMI".Btn_Ventilation_SCADA := FALSE;
   END_IF;
   //кнопка РОЗЖИГ на панели оператора
   "R_TRIG_DB_2"(CLK := "HMI".Btn_Ignition_HMI,
               Q => "FRONT_Btn_Ignition_HMI");
   IF "FRONT_Btn_Ignition_HMI" THEN
       "HMI".Btn_Ignition_HMI := FALSE;
   END_IF;
   //кнопка РОЗЖИГ на SCADA
   "R_TRIG_DB_3"(CLK := "HMI".Btn_Ignition_SCADA,
                 Q => "FRONT_Btn_Ignition_SCADA");
   IF "FRONT_Btn_Ignition_SCADA" THEN
       "HMI".Btn_Ignition_SCADA := FALSE;
   END_IF;
   //кнопка НОРМАЛЬНЫЙ ОСТАНОВ на панели оператора
   "R_TRIG_DB_4"(CLK := "HMI".Btn_normal_stop_HMI,
                 Q => "FRONT_Btn_Normal_stop_HMI");
   IF "FRONT_Btn_Normal_stop_HMI" THEN
       "HMI".Btn_normal_stop_HMI := FALSE;
   END_IF;
   //кнопка НОРМАЛЬНЫЙ ОСТАНОВ на SCADA
   "R_TRIG_DB_5"(CLK := "HMI".Btn_normal_stop_SCADA,
                 Q => "FRONT_Btn_Normal_stop_SCADA");
   IF "FRONT_Btn_Normal_stop_SCADA" THEN
       "HMI".Btn_normal_stop_SCADA := FALSE;
   END_IF;
   //кнопка АВАРИЙНЫЙ ОСТАНОВ на панели оператора
   "R_TRIG_DB_6"(CLK := "HMI".Btn_alarm_stop_HMI,
                 Q => "FRONT_Btn_Alarm_stop_HMI");
   IF "FRONT_Btn_Alarm_stop_HMI" THEN
       "HMI".Btn_alarm_stop_HMI := FALSE;
   END_IF;
   //кнопка АВАРИЙНЫЙ ОСТАНОВ на SCADA
   "R_TRIG_DB_7"(CLK := "HMI".Btn_alarm_stop_SCADA,
                 Q => "FRONT_Btn_Alarm_stop_SCADA");
   IF "FRONT_Btn_Alarm_stop_SCADA" THEN
       "HMI".Btn_alarm_stop_SCADA := FALSE;
   END_IF;
   //кнопка ТЕСТОВАЯ ОПРЕССОВКА на панели оператора
   "R_TRIG_DB_8"(CLK := "HMI".Btn_test_press_HMI,
                 Q => "FRONT_Btn_test_press_HMI");
   IF "FRONT_Btn_test_press_HMI" THEN
       "HMI".Btn_test_press_HMI := FALSE;
   END_IF;
   //кнопка ТЕСТОВЫЙ РОЗЖИГ на панели оператора
   "R_TRIG_DB_9"(CLK := "HMI".Btn_test_ignition_HMI,
                 Q => "FRONT_Btn_test_ignition_HMI");
   IF "FRONT_Btn_test_ignition_HMI" THEN
       "HMI".Btn_test_ignition_HMI := FALSE;
   END_IF;

   //кнопка РУЧНОЙ РОЗЖИГ на панели оператора
   (* "R_TRIG_DB_10"(CLK:="HMI".Btn_manual_ignition_HMI,
                  Q =>"FRONT_Btn_manual_ignition_HMI");
   IF "FRONT_Btn_manual_ignition_HMI" THEN
       "HMI".Btn_manual_ignition_HMI := FALSE;
   END_IF; *)
   IF NOT ("Technology".Regim = 3 AND "Technology".Regim_ventilation_step = 25) AND NOT ("Technology".Regim = 5 AND "Technology".Regim_ignition_step = 19) THEN
       "HMI".Btn_manual_ignition_HMI := FALSE;
   END_IF;

   //кнопка СБРОС ЗВУКА на панели оператора
   "R_TRIG_DB_28"(CLK := "HMI".Btn_reset_sound_HMI,
                 Q => "FRONT_Btn_reset_sound_HMI");
   IF "FRONT_Btn_reset_sound_HMI" THEN
       "HMI".Btn_reset_sound_HMI := FALSE;
   END_IF;

   (*Текущая уставка регулятора давления воздуха*)
   IF "Sensors".DV_invertor_mode.Value THEN
       "HMI".Current_SP_P_air :="Control_DV".SP_PID;
   END_IF;
   IF "Sensors".DV_powergrid_mode.Value THEN
       "HMI".Current_SP_P_air := "Control_NAV".SP_PID;
   END_IF;
   (*Текущая уставка регулятора разряжения*)
   IF "Sensors".DS_invertor_mode.Value THEN
       "HMI".Current_SP_dP_furnance := "Control_DS".SP_PID;
   END_IF;
   IF "Sensors".DS_powergrid_mode.Value THEN
       "HMI".Current_SP_dP_furnance := "Control_NAD".SP_PID;
   END_IF;

   (*Определение текущего подрежима*)
   CASE "Technology".Regim OF
       1:  //откл
           "HMI".INDICATION_TIME_1 := 255;
           "HMI".INDICATION_TIME_2 := 255;
           CASE "Technology".Regim_off_step OF
               0:  "Technology".Substage := 1; //перевод ИМ в дистанционный режим

               1:
                   "HMI".INDICATION_TIME_1 := 255;
                   "HMI".INDICATION_TIME_2 := 255;

                   IF "Message".VENTILATION_not_initial_state_air THEN
                       "Technology".Substage := 11; //НАД, НАВ не закрылись или не откл ДВ
                   ELSE
                       IF "Message".VENTILATION_NAV_not_close THEN
                           "Technology".Substage := 13; //НАВ не закрылся
                       ELSE
                           "Technology".Substage := 2; //ожидание нажатия кн.Вентиляция
                           //"Technology".Substage := 168; //ожидание дальнейших действий. Нажмите кн.Вентиляция или кн.Плановый останов
                       END_IF;
                   END_IF;

               2:
                   "HMI".INDICATION_TIME_1 := 255;
                   "HMI".INDICATION_TIME_2 := 255;
                   "Technology".Substage := 4; //перевод газовых клапанов в исходное положение

               3:
                   "HMI".INDICATION_TIME_1 := 255;
                   "HMI".INDICATION_TIME_2 := 255;
                   "Technology".Substage := 169; //отключение ДВ
               4:
                   "HMI".INDICATION_TIME_1 := 255;
                   "HMI".INDICATION_TIME_2 := 255;
                   "Technology".Substage := 170; //отключение ДС             
               ELSE
                   "Technology".Substage := 0; //неизвестно
           END_CASE;
       3:  //вентиляция
           CASE "Technology".Regim_ventilation_step OF
               0:
                   "HMI".INDICATION_TIME_1 := 255;
                   "HMI".INDICATION_TIME_2 := 255;
                   "Technology".Substage := 3; //проверка положения газовых клапанов (не используется)
               1:
                   "HMI".INDICATION_TIME_1 := 255;
                   "HMI".INDICATION_TIME_2 := 255;
                   IF NOT "Message".VENTILATION_not_initial_state_gas THEN
                       "Technology".Substage := 4; //перевод газовых клапанов в исходное положение
                   ELSE
                       "Technology".Substage := 5; //газовые клапана не перевелись в исходное положение
                   END_IF;
               2:
                   "HMI".INDICATION_TIME_1 := 255;
                   "HMI".INDICATION_TIME_2 := 255;
                   IF NOT "Message".VENTILATION_DS_need_dist_mode THEN
                       "Technology".Substage := 6; //проверка нахождения ШУД ДС в дистанционном режиме
                   ELSE
                       "Technology".Substage := 7; //необходимо перевести ШУД ДС в дистанционный режим
                   END_IF;
               3:
                   "HMI".INDICATION_TIME_1 := 255;
                   "HMI".INDICATION_TIME_2 := 255;
                   IF NOT "Message".VENTILATION_DV_need_dist_mode THEN
                       "Technology".Substage := 8; //проверка нахождения ШУД ДВ в дистанционном режиме
                   ELSE
                       "Technology".Substage := 9; //необходимо перевести ШУД ДВ в дистанционный режим
                   END_IF;
               4:
                   IF NOT "Message".VENTILATION_BRU_NAD_need_avto_mode THEN
                       "Technology".Substage := 171;   //проверка нахождения БРУ НАД в автоматическом режиме
                   ELSE
                       "Technology".Substage := 172;   //необходимо перевести БРУ НАД в автоматический режим
                   END_IF;
               5:
                   IF NOT "Message".VENTILATION_BRU_NAV_need_avto_mode THEN
                       "Technology".Substage := 173;   //проверка нахождения БРУ НАВ в автоматическом режиме
                   ELSE
                       "Technology".Substage := 174;   //необходимо перевести БРУ НАВ в автоматический режим
                   END_IF;
               6:
                   "HMI".INDICATION_TIME_1 := 255;
                   "HMI".INDICATION_TIME_2 := 255;
                   IF NOT "Message".VENTILATION_not_initial_state_air THEN
                       "Technology".Substage := 10; //закрытие НАД, НАВ, откл ДВ
                   ELSE
                       "Technology".Substage := 11; //НАД, НАВ не закрылись или не откл ДВ
                   END_IF;
               7:
                   "HMI".INDICATION_TIME_1 := 255;
                   "HMI".INDICATION_TIME_2 := 255;
                   IF NOT "Message".VENTILATION_NAV_not_close THEN
                       "Technology".Substage := 12; //закрытие НАВ
                   ELSE
                       "Technology".Substage := 13; //НАВ не закрылся
                   END_IF;
               8:
                   "HMI".INDICATION_TIME_1 := 255;
                   "HMI".INDICATION_TIME_2 := 255;
                   "Technology".Substage := 14; //проверка состояния ДС
               9:
                   "HMI".INDICATION_TIME_1 := 255;
                   "HMI".INDICATION_TIME_2 := 255;
                   IF NOT "Message".VENTILATION_DS_not_on THEN
                       "Technology".Substage := 15; //пуск ДС
                   ELSE
                       "Technology".Substage := 16; //ДС не включился
                   END_IF;
               10:
                   "HMI".INDICATION_TIME_1 := 255;
                   "HMI".INDICATION_TIME_2 := 255;
                   "Technology".Substage := 15; //пуск ДС
               11:
                   "HMI".INDICATION_TIME_1 := 255;
                   "HMI".INDICATION_TIME_2 := 255;
                   "Technology".Substage := 17; //проверка состояния ДВ
               12:
                   "HMI".INDICATION_TIME_1 := 255;
                   "HMI".INDICATION_TIME_2 := 255;
                   IF NOT "Message".VENTILATION_DV_not_on THEN
                       "Technology".Substage := 18; //пуск ДВ
                   ELSE
                       "Technology".Substage := 19; //ДВ не включился
                   END_IF;
               13:
                   "HMI".INDICATION_TIME_1 := 255;
                   "HMI".INDICATION_TIME_2 := 255;
                   "Technology".Substage := 18; //пуск ДВ
               14:
                   "HMI".INDICATION_TIME_1 := 255;
                   "HMI".INDICATION_TIME_2 := 255;
                   IF NOT "Message".VENTILATION_NAD_not_open_manual THEN
                       "Technology".Substage := 20; //открытие НАД
                   ELSE
                       "Technology".Substage := 21; //БРУ НАД в местром режиме и НАД не открыт
                   END_IF;
                   (* IF NOT "Message".VENTILATION_NAD_not_open THEN
                       "Technology".Substage := 20; //открытие НАД
                   ELSE
                       "Technology".Substage := 21; //НАД не открылся
                   END_IF; *)
               15:
                   "HMI".INDICATION_TIME_1 := 255;
                   "HMI".INDICATION_TIME_2 := 255;
                   "Technology".Substage := 20; //открытие НАД
               16:
                   "HMI".INDICATION_TIME_1 := 255;
                   "HMI".INDICATION_TIME_2 := 255;

                   IF NOT "Message".VENTILATION_NAV_not_open_manual THEN
                       IF NOT "Message".VENTILATION_NAV_or_NAD_not_open THEN
                           "Technology".Substage := 22; //открытие НАВ и НАД
                       ELSE
                           "Technology".Substage := 23; //НАВ или НАД не открылись
                       END_IF;
                   ELSE
                       "Technology".Substage := 33; //БРУ НАВ в местром режиме и НАВ не открыт
                   END_IF;
               17:
                   "HMI".INDICATION_TIME_1 := 255;
                   "HMI".INDICATION_TIME_2 := 255;
                   "Technology".Substage := 22; //открытие НАВ и НАД
               18:
                   "HMI".INDICATION_TIME_1 := 255;
                   "HMI".INDICATION_TIME_2 := 255;
                   "Technology".Substage := 24; //Включаем ПИД ДС на вентиляционные параметры
               19:
                   "HMI".INDICATION_TIME_1 := 255;
                   "HMI".INDICATION_TIME_2 := 255;
                   "Technology".Substage := 24; //Включаем ПИД ДС на вентиляционные параметры
               20:
                   "HMI".INDICATION_TIME_1 := 255;
                   "HMI".INDICATION_TIME_2 := 255;
                   "Technology".Substage := 25; //Включаем ПИД ДВ на вентиляционные параметры
               21:
                   "HMI".INDICATION_TIME_1 := 255;
                   "HMI".INDICATION_TIME_2 := 255;
                   "Technology".Substage := 25; //Включаем ПИД ДВ на вентиляционные параметры
               22:
                   "HMI".INDICATION_TIME_1 := 255;
                   "HMI".INDICATION_TIME_2 := 255;
                   "Technology".Substage := 26; //Проверка достижения вентиляционных параметров
               23:
                   "HMI".TIME_converter_IN := "Timer_VENTILATION_DB".PT -"Timer_VENTILATION_DB".ET;
                   "HMI".INDICATION_TIME_1 := INT_TO_USINT("HMI".TIME_converter_minute);
                   "HMI".INDICATION_TIME_2 := INT_TO_USINT("HMI".TIME_converter_second);

                   IF "Message".VENTILATION_run THEN
                       "Technology".Substage := 27; //вентиляция топки
                   ELSE
                       "Technology".Substage := 28; //параметры вентиляции не в норме
                   END_IF;
               24:
                   "HMI".INDICATION_TIME_1 := 255;
                   "HMI".INDICATION_TIME_2 := 255;
                   "Technology".Substage := 29; //вентиляция прервана. Устраните неисправность. Для повторного проведения нажмите кн.Вентиляция. Для останова нажмите кн.Плановый останов
               25:
                   "HMI".INDICATION_TIME_1 := 255;
                   "HMI".INDICATION_TIME_2 := 255;
                   IF NOT "Message".VENTILATION_Check_param THEN
                       IF NOT "Message".TEST_PRESS_ok THEN
                           "Technology".Substage := 30; //вентиляция проведена. Ожидание дальнейших действий
                       ELSE
                           "Technology".Substage := 31; //тестовая опрессовка успешно проведена
                       END_IF;
                   ELSE
                       "Technology".Substage := 32; //переход невозможен. Проверьте параметры вентиляции
                   END_IF;
               ELSE
                   "HMI".INDICATION_TIME_1 := 255;
                   "HMI".INDICATION_TIME_2 := 255;
                   "Technology".Substage := 0; //неизвестно
           END_CASE;
       4:  //опрессовка
           "HMI".INDICATION_TIME_1 := 255;
           "HMI".INDICATION_TIME_2 := 255;
           CASE "Technology".Regim_press_step OF
               0:
                   "Technology".Substage := 40; //открытие ЗДСВ
               1:
                   "Technology".Substage := 41; //перевод регулятора разрежения на розжиговые параметры
               2:
                   "Technology".Substage := 42; //перевод регулятора разрежения на розжиговые параметры
               3:
                   "Technology".Substage := 43; //перевод регулятора давления воздуха на розжиговые параметры
               4:
                   "Technology".Substage := 44; //перевод регулятора давления воздуха на розжиговые параметры
               5:
                   "Technology".Substage := 45; //проверка достижения розжиговых параметров
               6:
                   IF NOT "Message".PRESS_not_initial_state_gas THEN
                       "Technology".Substage := 46; //перевод клапанов по газу в исходное состояние
                   ELSE
                       "Technology".Substage := 47; //клапана по газу не переведены в исходное состояние
                   END_IF;
               7:
                   IF NOT "Message".PRESS_ZRG_not_close THEN
                       "Technology".Substage := 48; //закрываем ЗРГ
                   ELSE
                       "Technology".Substage := 49; //ЗРГ не закрылся
                   END_IF;
               8:
                   IF NOT "Message".PRESS_ZDG_not_open THEN
                       "Technology".Substage := 50; //открываем ЗДГ
                   ELSE
                       "Technology".Substage := 51; //ЗДГ не открылся
                   END_IF;
               9:
                   "Technology".Substage := 52; //заполнение газом
               10:
                   "Technology".Substage := 53; //контроль давления перед БГ
               11:
                   "Technology".Substage := 54; //давления перед БГ не в норме. Устраните неисправность. Для продолжения нажмите кн.Розжиг
               12:
                   "Technology".Substage := 55; //проверка давления между ПЗК с открытым КБ
               13:
                   "Technology".Substage := 56; //проверка давления между ПЗК с закрытым КБ
               14:
                   "Technology".Substage := 57; //проверка на MIN. Открытие КО 
               15:
                   "Technology".Substage := 58; //проверка на MIN
               16:    
                   "Technology".Substage := 58; //проверка на MIN
               17:
                   "Technology".Substage := 59; //проверка на MAX. Открытие КБ
               18:
                   "Technology".Substage := 59; //проверка на MAX. Открытие КБ
               19:
                   "Technology".Substage := 60; //проверка на MAX. Открытие КО
               20:
                   "Technology".Substage := 61; //проверка на MAX
               21:
                   "Technology".Substage := 62; //проверка на MAX
               22:
                   IF "Message".PRESS_not_initial_state_gas THEN
                       "Technology".Substage := 63; //Механизмы по газу не переведены в исходное состояние. Устраните неисправность и для продолжения нажмите кн.Розжиг
                   END_IF;
                   IF "Message".PRESS_PZK1_or_KO_untight THEN
                       "Technology".Substage := 64; //ПЗК1 или КО неплотен. Устраните неисправность и для продолжения нажмите кн.Розжиг
                   END_IF;
                   IF "Message".PRESS_Not_orifice_plate_or_PZK1_untight THEN
                       "Technology".Substage := 65; //нет дроссельной шайбы или ПЗК1 неплотен. Устраните неисправность и для продолжения нажмите кн.Розжиг
                   END_IF;
                   IF "Message".PRESS_PZK2_or_KB_untight THEN
                       "Technology".Substage := 66; //ПЗК2 или КБ неплотен. Устраните неисправность и для продолжения нажмите кн.Розжиг
                   END_IF;
               23:
                   "Technology".Substage := 175; //опрессовка успешно проведена
               ELSE
                   "Technology".Substage := 0; //неизвестно
           END_CASE;
       5:  //розжиг
           "HMI".INDICATION_TIME_1 := 255;
           "HMI".INDICATION_TIME_2 := 255;
           CASE "Technology".Regim_ignition_step OF
               0:
                   IF NOT "Message".IGNITION_ZRG_not_close THEN
                       "Technology".Substage := 70; //закрываем ЗРГ
                   ELSE
                       "Technology".Substage := 71; //ЗРГ не закрылся
                   END_IF;
               1:
                   IF NOT "Message".IGNITION_PZK2_not_close THEN
                       "Technology".Substage := 72; //контроль закрытого положения ПЗК2
                   ELSE
                       "Technology".Substage := 73; //ПЗК2 не закрыт
                   END_IF;
               2:
                   IF NOT "Message".IGNITION_KZ_not_close THEN
                       "Technology".Substage := 74; //контроль закрытого положения КЗ
                   ELSE
                       "Technology".Substage := 75; //КЗ не закрыт
                   END_IF;
               3:
                   IF NOT "Message".IGNITION_KB_not_close THEN
                       "Technology".Substage := 76; //закрываем КБ
                   ELSE
                       "Technology".Substage := 77; //КБ не закрылся
                   END_IF;
               4:
                   "Technology".Substage := 76; //закрываем КБ
               5:
                   IF NOT "Message".IGNITION_PZK1_not_open THEN
                       "Technology".Substage := 78; //открываем ПЗК1
                   ELSE
                       "Technology".Substage := 79; //ПЗК1 не открылся
                   END_IF;

               6:
                   "Technology".Substage := 78; //открываем ПЗК1
               7:
                   "Technology".Substage := 80; //включаем ИВН
               8:
                   IF "Technology".CNT_Igniter = 1 THEN
                       "Technology".Substage := 81; //включаем ИВН. 1 попытка розжига запальника
                   END_IF;
                   IF "Technology".CNT_Igniter = 2 THEN
                       "Technology".Substage := 82; //включаем ИВН. 2 попытка розжига запальника
                   END_IF;
               9:
                   IF "Technology".CNT_Igniter = 1 THEN
                       IF NOT "Message".IGNITION_KZ_not_open THEN
                           "Technology".Substage := 83; //открываем КЗ. 1 попытка розжига запальника
                       ELSE
                           "Technology".Substage := 84; //КЗ не открылся. 1 попытка розжига запальника
                       END_IF;
                   END_IF;
                   IF "Technology".CNT_Igniter = 2 THEN
                       IF NOT "Message".IGNITION_KZ_not_open THEN
                           "Technology".Substage := 85; //открываем КЗ. 2 попытка розжига запальника
                       ELSE
                           "Technology".Substage := 86; //КЗ не открылся. 2 попытка розжига запальника
                       END_IF;
                   END_IF;
               10:
                   IF "Technology".CNT_Igniter = 1 THEN
                       "Technology".Substage := 87; //розжиг запальника 1 попытка
                   END_IF;
                   IF "Technology".CNT_Igniter = 2 THEN
                       "Technology".Substage := 88; //розжиг запальника 2 попытка
                   END_IF;
               11:
                   IF "Technology".CNT_Igniter = 1 THEN
                       "Technology".Substage := 89; //контроль пламени запальника. 1 попытка розжига
                   END_IF;
                   IF "Technology".CNT_Igniter = 2 THEN
                       "Technology".Substage := 90; //контроль пламени запальника. 2 попытка розжига
                   END_IF;
               12:
                   "Technology".Substage := 91; //запальник не разжегся. Перевод клапанов в исходное положение
               13:
                   IF NOT "Message".IGNITION_not_initial_state_gas THEN
                       "Technology".Substage := 92; //запальник не разжегся. Для повторной попытки нажмите кн. РОЗЖИГ
                   ELSE
                       "Technology".Substage := 93; //газовые клапана не переведены в исходное состояние
                   END_IF;
               14:
                   "Technology".Substage := 94; //открываем ПЗК2
               15:
                   "Technology".Substage := 95; //розжиг горелки
               16:
                   "Technology".Substage := 96; //розжиг горелки
               17:
                   "Technology".Substage := 97; //стабилизация пламени горелки
               18:
                   IF "Sensors".KZ_control_open.Value THEN
                       "Technology".Substage := 98; //ожидание закрытия КЗ
                   ELSE
                       IF "Message".TEST_IGNITION_ok THEN
                           "Technology".Substage := 99; //тестовый розжиг успешно произведен
                       END_IF;
                   END_IF;
               19:
                   "Technology".Substage := 100; //режим ручного розжига
               20:
                   "Technology".Substage := 88; //розжиг запальника 2 попытка
               21:
                   "Technology".Substage := 88; //розжиг запальника 2 попытка
               ELSE
                   "Technology".Substage := 0; //неизвестно
           END_CASE;
       6:  //выход на MIN мощность
           "HMI".INDICATION_TIME_1 := 255;
           "HMI".INDICATION_TIME_2 := 255;
           CASE "Technology".Regim_min_power_step OF
               0:
                   "Technology".Substage := 110; //переводим ПИД разряжения на работу по режимной карте
               1:
                   "Technology".Substage := 111; //переводим ПИД разряжения на работу по режимной карте
               2:
                   "Technology".Substage := 112; //переводим ПИД давления воздуха на работу по режимной карте
               3:
                   "Technology".Substage := 113; //переводим ПИД давления воздуха на работу по режимной карте
               4:
                   "Technology".Substage := 114; //открываем ЗРГ до значения минимальной мощности
               ELSE
                   "Technology".Substage := 0; //неизвестно
           END_CASE;
       7:  //прогрев
           CASE "Technology".Regim_heating_step OF
               0:
                   "HMI".INDICATION_TIME_1 := 255;
                   "HMI".INDICATION_TIME_2 := 255;
                   "Technology".Substage := 115; //переводим ЗРГ в дистанционный режим
               1:
                   "HMI".TIME_converter_IN := "Timer_HEATING_temp_DB".PT - "Timer_HEATING_temp_DB".ET;
                   "HMI".INDICATION_TIME_1 := INT_TO_USINT("HMI".TIME_converter_minute);
                   "HMI".INDICATION_TIME_2 := INT_TO_USINT("HMI".TIME_converter_second);

                   "Technology".Substage := 116; //процесс прогрева
               ELSE
                   "HMI".INDICATION_TIME_1 := 255;
                   "HMI".INDICATION_TIME_2 := 255;
                   "Technology".Substage := 0; //неизвестно
           END_CASE;
       8:  //работа
           CASE "Technology".Regim_run_step OF
               0:
                   IF NOT "Protections".BLOCK_Not_flame_burner THEN
                       "HMI".LTIME_converter_IN := "Timer_RUN_temp_DB".ET;
                       "HMI".INDICATION_TIME_1 := DINT_TO_USINT("HMI".LTIME_converter_day);
                       "HMI".INDICATION_TIME_2 := INT_TO_USINT("HMI".LTIME_converter_hour);
                   ELSE    //если имеется блокировка защиты по погасанию пламени горелки
                       "HMI".TIME_converter_IN := "TON_protection_13_DB".PT - "TON_protection_13_DB".ET;
                       "HMI".INDICATION_TIME_1 := INT_TO_USINT("HMI".TIME_converter_minute);
                       "HMI".INDICATION_TIME_2 := INT_TO_USINT("HMI".TIME_converter_second);
                   END_IF;
                   "Technology".Substage := 117; //процесс работы 
               ELSE
                   "HMI".INDICATION_TIME_1 := 255;
                   "HMI".INDICATION_TIME_2 := 255;
                   "Technology".Substage := 0; //неизвестно
           END_CASE;
       9:  //экстренный останов
           "HMI".INDICATION_TIME_1 := 255;
           "HMI".INDICATION_TIME_2 := 255;
           CASE "Technology".Regim_emergency_stop_step OF
               0:
                   IF NOT "Message".EMERGENCY_STOP_not_initial_state THEN
                       "Technology".Substage := 120; //отключение всего 
                   ELSE
                       "Technology".Substage := 121; //устройства не переведены в исходное состояние
                   END_IF;
               ELSE
                   "Technology".Substage := 0; //неизвестно
           END_CASE;
       10: //аварийный останов
           "HMI".INDICATION_TIME_1 := 255;
           "HMI".INDICATION_TIME_2 := 255;
           CASE "Technology".Regim_alarm_stop_step OF
               0:
                   IF NOT "Message".ALARM_STOP_not_initial_state_gas THEN
                       "Technology".Substage := 122; //перевод всех газовых клапанов в исходное состояние
                   ELSE
                       "Technology".Substage := 123; //газовые клапана не переведены в исходное состояние
                   END_IF;
               ELSE
                   "Technology".Substage := 0; //неизвестно
           END_CASE;
       11: //плановый останов
           "HMI".INDICATION_TIME_1 := 255;
           "HMI".INDICATION_TIME_2 := 255;
           CASE "Technology".Regim_plan_stop_step OF
               0:
                   "Technology".Substage := 130; //вывод ЗРГ на значение минимальной мощности
               1:
                   "Technology".Substage := 131; //вывод ЗРГ на значение минимальной мощности
               2:
                   IF NOT "Message".PLAN_STOP_not_initial_state_gas THEN
                       "Technology".Substage := 132; //перевод газовых клапанов в исходное состояние, регуляторов разряжения и вентиляции на вентиляционные параметры
                   ELSE
                       "Technology".Substage := 133; //газовые клапана не переведены в исходное состояние
                   END_IF;
               3:
                   "Technology".Substage := 134; //перевод регуляторов разряжения и вентиляции на вентиляционные параметры
               ELSE
                   "Technology".Substage := 0; //неизвестно
           END_CASE;
       12: //постостановочная опрессовка
           "HMI".INDICATION_TIME_1 := 255;
           "HMI".INDICATION_TIME_2 := 255;
           CASE "Technology".Regim_stop_press_step OF
               0:
                   "Technology".Substage := 140; //анализ разрешения проведения постостановочной опрессовки
               1:
                   "Technology".Substage := 141; //контроль положения исполнительных механизмов по газу
               2:
                   "Technology".Substage := 142; //контроль min P
               3:
                   "Technology".Substage := 143; //контроль max P
               4:
                   "Technology".Substage := 144; //закрываем КБ
               5:
                   "Technology".Substage := 145; //контроль отсутствия давления газа м/у ПЗК
               6:
                   "Technology".Substage := 146; //открываем КО
               7:
                   "Technology".Substage := 147; //контроль достижения давления газа м/у ПЗК
               8:
                   "Technology".Substage := 148; //закрываем КО
               9:
                   "Technology".Substage := 149; //открываем КБ
               10:
                   "Technology".Substage := 150; //определение успешности постостановочной опрессовки
               11:
                   IF "Message".STOP_PRESS_PZK1_or_KO_untight THEN
                       "Technology".Substage := 151; //постостановочная опрессовка не прошла. ПЗК1 или КО негерметичен
                   END_IF;
                   IF "Message".STOP_PRESS_PZK2_or_KB_untight THEN
                       "Technology".Substage := 152; //постостановочная опрессовка не прошла. ПЗК2 или КБ негерметичен
                   END_IF;
                   IF "Message".STOP_PRESS_P_before_BG_min THEN
                       "Technology".Substage := 153; //постостановочная опрессовка не прошла. Низкое давление до БГ
                   END_IF;
                   IF "Message".STOP_PRESS_success THEN
                       "Technology".Substage := 154; //постостановочная опрессовка успешно проведена
                   END_IF;
               ELSE
                   "Technology".Substage := 0; //неизвестно
           END_CASE;
       13: //укороченная вентиляция
           CASE "Technology".Regim_short_ventilation_step OF
               0:
                   "HMI".INDICATION_TIME_1 := 255;
                   "HMI".INDICATION_TIME_2 := 255;
                   "Technology".Substage := 160; //анализ необходимости проведения укороченной вентиляции
               1:
                   "HMI".INDICATION_TIME_1 := 255;
                   "HMI".INDICATION_TIME_2 := 255;
                   "Technology".Substage := 161; //переход на поддержание вентиляционного значения разрежения
               2:
                   "HMI".INDICATION_TIME_1 := 255;
                   "HMI".INDICATION_TIME_2 := 255;
                   "Technology".Substage := 162; //переход на поддержание вентиляционного значения разрежения
               3:
                   "HMI".INDICATION_TIME_1 := 255;
                   "HMI".INDICATION_TIME_2 := 255;
                   "Technology".Substage := 163; //переход на поддержание вентиляционного значения давления воздуха
               4:
                   "HMI".TIME_converter_IN := "Timer_SHORT_VENTILATION_temp_DB".PT - "Timer_SHORT_VENTILATION_temp_DB".ET;
                   "HMI".INDICATION_TIME_1 := INT_TO_USINT("HMI".TIME_converter_minute);
                   "HMI".INDICATION_TIME_2 := INT_TO_USINT("HMI".TIME_converter_second);
                   "Technology".Substage := 164; //процесс вентиляции
               5:
                   "HMI".INDICATION_TIME_1 := 255;
                   "HMI".INDICATION_TIME_2 := 255;
                   "Technology".Substage := 165; //переход на поддержание розжигового значения разрежения
               6:
                   "HMI".INDICATION_TIME_1 := 255;
                   "HMI".INDICATION_TIME_2 := 255;
                   "Technology".Substage := 166; //переход на поддержание розжигового значения разрежения
               7:
                   "HMI".INDICATION_TIME_1 := 255;
                   "HMI".INDICATION_TIME_2 := 255;
                   "Technology".Substage := 167; //переход на поддержание розжигового значения давления воздуха
               ELSE
                   "HMI".INDICATION_TIME_1 := 255;
                   "HMI".INDICATION_TIME_2 := 255;
                   "Technology".Substage := 0; //неизвестно
           END_CASE;
       ELSE
           "Technology".Substage := 0; //неизвестно
   END_CASE;

   "TIME_converter_DB"(IN := "HMI".TIME_converter_IN,
                       Minute => "HMI".TIME_converter_minute,
                       Second => "HMI".TIME_converter_second);

   "LTIME_converter_DB"(IN := "HMI".LTIME_converter_IN,
                        Day=>"HMI".LTIME_converter_day,
                        Hour=>"HMI".LTIME_converter_hour);
END_FUNCTION

FUNCTION "Log" : Void   // FC29, SCL
{ S7_Optimized_Access := 'TRUE' }
VERSION : 0.1
BEGIN
   (*Нажатие кнопок для журнала событий*)
   (*Кнопка ВЕНТИЛЯЦИЯ на панели оператора для журнала событий*)
   IF "HMI".Btn_Ventilation_HMI THEN
       "HMI".Btn_Ventilation_HMI_Log := TRUE;
   END_IF;
   (*Кнопка ВЕНТИЛЯЦИЯ на SCADA для журнала событий*)
   IF "HMI".Btn_Ventilation_SCADA THEN
       "HMI".Btn_Ventilation_SCADA_Log := TRUE;
   END_IF;
   (*Кнопка ВЕНТИЛЯЦИЯ на ШАУ для журнала событий*)
   IF "Sensors".Btn_Ventilation.Value THEN
       "HMI".Btn_Ventilation_ShAU_Log := TRUE;
   END_IF;
   (*Кнопка РОЗЖИГ на панели оператора для журнала событий*)
   IF "HMI".Btn_Ignition_HMI THEN
       "HMI".Btn_Ignition_HMI_Log := TRUE;
   END_IF;
   (*Кнопка РОЗЖИГ на SCADA для журнала событий*)
   IF "HMI".Btn_Ignition_SCADA THEN
       "HMI".Btn_Ignition_SCADA_Log := TRUE;
   END_IF;
   (*Кнопка РОЗЖИГ на ШАУ для журнала событий*)
   IF "Sensors".Btn_Ignition.Value THEN
       "HMI".Btn_Ignition_ShAU_Log := TRUE;
   END_IF;
   (*Кнопка НОРМАЛЬНЫЙ ОСТАНОВ на панели оператора для журнала событий*)
   IF "HMI".Btn_normal_stop_HMI THEN
       "HMI".Btn_normal_stop_HMI_Log := TRUE;
   END_IF;
   (*Кнопка НОРМАЛЬНЫЙ ОСТАНОВ на SCADA для журнала событий*)
   IF "HMI".Btn_normal_stop_SCADA THEN
       "HMI".Btn_normal_stop_SCADA_Log := TRUE;
   END_IF;
   (*Кнопка АВАРИЙНЫЙ ОСТАНОВ на панели оператора для журнала событий*)
   IF "HMI".Btn_alarm_stop_HMI THEN
       "HMI".Btn_alarm_stop_HMI_Log := TRUE;
   END_IF;
   (*Кнопка АВАРИЙНЫЙ ОСТАНОВ на SCADA для журнала событий*)
   IF "HMI".Btn_alarm_stop_SCADA THEN
       "HMI".Btn_alarm_stop_SCADA_Log := TRUE;
   END_IF;
   (*Кнопка ЭКСТРЕННЫЙ ОСТАНОВ на ШАУ для журнала событий*)
   IF "Sensors".Btn_STOP.Value THEN
       "HMI".Btn_emergency_stop_ShAU_Log := TRUE;
   END_IF;
   (*Кнопка ТЕСТОВАЯ ОПРЕССОВКА на панели оператора для журнала событий*)
   IF "HMI".Btn_test_press_HMI THEN
       "HMI".Btn_test_press_HMI_Log := TRUE;
   END_IF;
   (*Кнопка ТЕСТОВЫЙ РОЗЖИГ на панели оператора для журнала событий*)
   IF "HMI".Btn_test_ignition_HMI THEN
       "HMI".Btn_test_ignition_HMI_Log := TRUE;
   END_IF;
   (*Кнопка Ручной РОЗЖИГ на панели оператора для журнала событий*)
   IF "HMI".Btn_manual_ignition_HMI THEN
       "HMI".Btn_manual_ignition_HMI_Log := TRUE;
   END_IF;
   (*Кнопка СБРОС ЗВУКА на панели оператора для журнала событий*)
   IF "HMI".Btn_reset_sound_HMI THEN
       "HMI".Btn_reset_sound_HMI_Log := TRUE;
   END_IF;
   (*(*СБРОС аварий для журнала событий*)
   IF "Alarms_and_warnings".Reset_alarms THEN
       "HMI".Reset_alarms_Log := TRUE;
   END_IF;*)
   (*СБРОС аварий на ШАУ для журнала событий*)
   IF "Sensors".Btn_Sound.Value THEN
       "HMI".Btn_reset_alarms_ShAU_Log := TRUE;
   END_IF;
   (*(*Режимная карта. Применить. Для журнала событий*)
   IF "RegMap".Apply THEN
       "HMI".RegMap_Apply_Log := TRUE;
   END_IF;*)
   (*(*ДС. Ручное управление. Пуск. Для журнала событий*)
   IF "Control_DS".Manual_Start THEN
       "HMI".DS_Manual_Start_Log := TRUE;
   END_IF;
   (*ДС. Ручное управление. Стоп. Для журнала событий*)
   IF "Control_DS".Manual_Stop THEN
       "HMI".DS_Manual_Stop_Log := TRUE;
   END_IF;
   (*ДВ. Ручное управление. Пуск. Для журнала событий*)
   IF "Control_DV".Manual_Start THEN
       "HMI".DV_Manual_Start_Log := TRUE;
   END_IF;
   (*ДВ. Ручное управление. Стоп. Для журнала событий*)
   IF "Control_DV".Manual_Stop THEN
       "HMI".DV_Manual_Stop_Log := TRUE;
   END_IF;
   (*ЗДГ. Ручное управление. Открыть. Для журнала событий*)
   IF "Control_ZDG".Manual_open THEN
       "HMI".ZDG_Manual_open_Log := TRUE;
   END_IF;
   (*ЗДГ. Ручное управление. Закрыть. Для журнала событий*)
   IF "Control_ZDG".Manual_close THEN
       "HMI".ZDG_Manual_close_Log := TRUE;
   END_IF;
   (*ЗДГ. Ручное управление. Стоп. Для журнала событий*)
   IF "Control_ZDG".Manual_stop THEN
       "HMI".ZDG_Manual_stop_Log := TRUE;
   END_IF;
   (*ЗДСВ после котла. Ручное управление. Открыть. Для журнала событий*)
   IF "Control_ZDSV_after_boiler".Manual_open THEN
       "HMI".ZDSV_after_boiler_Manual_open_Log := TRUE;
   END_IF;
   (*ЗДСВ после котла. Ручное управление. Закрыть. Для журнала событий*)
   IF "Control_ZDSV_after_boiler".Manual_close THEN
       "HMI".ZDSV_after_boiler_Manual_close_Log := TRUE;
   END_IF;
   (*ЗДСВ после котла. Ручное управление. Стоп. Для журнала событий*)
   IF "Control_ZDSV_after_boiler".Manual_stop THEN
       "HMI".ZDSV_after_boiler_Manual_stop_Log := TRUE;
   END_IF;
   (*ЗДСВ перед котлом. Ручное управление. Открыть. Для журнала событий*)
   IF "Control_ZDSV_before_boiler".Manual_open THEN
       "HMI".ZDSV_before_boiler_Manual_open_Log := TRUE;
   END_IF;
   (*ЗДСВ перед котлом. Ручное управление. Закрыть. Для журнала событий*)
   IF "Control_ZDSV_before_boiler".Manual_close THEN
       "HMI".ZDSV_before_boiler_Manual_close_Log := TRUE;
   END_IF;
   (*ЗДСВ перед котлом. Ручное управление. Стоп. Для журнала событий*)
   IF "Control_ZDSV_before_boiler".Manual_stop THEN
       "HMI".ZDSV_before_boiler_Manual_stop_Log := TRUE;
   END_IF;*)

   IF "HMI".Btn_Ventilation_HMI OR
       "HMI".Btn_Ventilation_SCADA OR
       "Sensors".Btn_Ventilation.Value OR
       "HMI".Btn_Ignition_HMI OR
       "HMI".Btn_Ignition_SCADA OR
       "Sensors".Btn_Ignition.Value OR
       "HMI".Btn_normal_stop_HMI OR
       "HMI".Btn_normal_stop_SCADA OR
       "HMI".Btn_alarm_stop_HMI OR
       "HMI".Btn_alarm_stop_SCADA OR
       "Sensors".Btn_STOP.Value OR
       "HMI".Btn_test_press_HMI OR
       "HMI".Btn_test_ignition_HMI OR
       "HMI".Btn_manual_ignition_HMI OR
       "HMI".Btn_reset_sound_HMI OR
       "Alarms_and_warnings".Reset_alarms OR
       "Sensors".Btn_Sound.Value OR
       "RegMap".Apply OR
       "Control_DS".Manual_Start OR
       "Control_DS".Manual_Stop OR
       "Control_DV".Manual_Start OR
       "Control_DV".Manual_Stop OR
       "Control_ZDG".Manual_open OR
       "Control_ZDG".Manual_close OR
       "Control_ZDG".Manual_stop OR
       "Control_ZDSV_after_boiler".Manual_open OR
       "Control_ZDSV_after_boiler".Manual_close OR
       "Control_ZDSV_after_boiler".Manual_stop OR
       "Control_ZDSV_before_boiler".Manual_open OR
       "Control_ZDSV_before_boiler".Manual_close OR
       "Control_ZDSV_before_boiler".Manual_stop THEN
       "Timer".Log_IN := TRUE;
   END_IF;

   IF NOT "HMI".Btn_Ventilation_HMI AND
       NOT "HMI".Btn_Ventilation_SCADA AND
       NOT "Sensors".Btn_Ventilation.Value AND
       NOT "HMI".Btn_Ignition_HMI AND
       NOT "HMI".Btn_Ignition_SCADA AND
       NOT "Sensors".Btn_Ignition.Value AND
       NOT "HMI".Btn_normal_stop_HMI AND
       NOT "HMI".Btn_normal_stop_SCADA AND
       NOT "HMI".Btn_alarm_stop_HMI AND
       NOT "HMI".Btn_alarm_stop_SCADA AND
       NOT "Sensors".Btn_STOP.Value AND
       NOT "HMI".Btn_test_press_HMI AND
       NOT "HMI".Btn_test_ignition_HMI AND
       NOT "HMI".Btn_manual_ignition_HMI AND
       NOT "HMI".Btn_reset_sound_HMI AND
       NOT "Alarms_and_warnings".Reset_alarms AND
       NOT "Sensors".Btn_Sound.Value AND
       NOT "RegMap".Apply AND
       NOT "Control_DS".Manual_Start AND
       NOT "Control_DS".Manual_Stop AND
       NOT "Control_DV".Manual_Start AND
       NOT "Control_DV".Manual_Stop AND
       NOT "Control_ZDG".Manual_open AND
       NOT "Control_ZDG".Manual_close AND
       NOT "Control_ZDG".Manual_stop AND
       NOT "Control_ZDSV_after_boiler".Manual_open AND
       NOT "Control_ZDSV_after_boiler".Manual_close AND
       NOT "Control_ZDSV_after_boiler".Manual_stop AND
       NOT "Control_ZDSV_before_boiler".Manual_open AND
       NOT "Control_ZDSV_before_boiler".Manual_close AND
       NOT "Control_ZDSV_before_boiler".Manual_stop THEN
       "Timer".Log_IN := FALSE;
   END_IF;

   "TOF_Log_DB".TOF(IN := "Timer".Log_IN,
                    PT := "Timer".Log_PT,
                    Q => "Timer".Log_Q);

   IF NOT "Timer".Log_Q THEN
       "HMI".Btn_Ventilation_HMI_Log := FALSE;
       "HMI".Btn_Ventilation_SCADA_Log := FALSE;
       "HMI".Btn_Ventilation_ShAU_Log := FALSE;
       "HMI".Btn_Ignition_HMI_Log := FALSE;
       "HMI".Btn_Ignition_SCADA_Log := FALSE;
       "HMI".Btn_Ignition_ShAU_Log := FALSE;
       "HMI".Btn_normal_stop_HMI_Log := FALSE;
       "HMI".Btn_normal_stop_SCADA_Log := FALSE;
       "HMI".Btn_alarm_stop_HMI_Log := FALSE;
       "HMI".Btn_alarm_stop_SCADA_Log := FALSE;
       "HMI".Btn_emergency_stop_ShAU_Log := FALSE;
       "HMI".Btn_test_press_HMI_Log := FALSE;
       "HMI".Btn_test_ignition_HMI_Log := FALSE;
       "HMI".Btn_manual_ignition_HMI_Log := FALSE;
       "HMI".Btn_reset_sound_HMI_Log := FALSE;
       "HMI".Reset_alarms_Log := FALSE;
       "HMI".Btn_reset_alarms_ShAU_Log := FALSE;
       "HMI".RegMap_Apply_Log := FALSE;
       "HMI".DS_Manual_Start_Log := FALSE;
       "HMI".DS_Manual_Stop_Log := FALSE;
       "HMI".DV_Manual_Start_Log := FALSE;
       "HMI".DV_Manual_Stop_Log := FALSE;
       "HMI".ZDG_Manual_open_Log := FALSE;
       "HMI".ZDG_Manual_close_Log := FALSE;
       "HMI".ZDG_Manual_stop_Log := FALSE;
       "HMI".ZDSV_after_boiler_Manual_open_Log := FALSE;
       "HMI".ZDSV_after_boiler_Manual_close_Log := FALSE;
       "HMI".ZDSV_after_boiler_Manual_stop_Log := FALSE;
       "HMI".ZDSV_before_boiler_Manual_open_Log := FALSE;
       "HMI".ZDSV_before_boiler_Manual_close_Log := FALSE;
       "HMI".ZDSV_before_boiler_Manual_stop_Log := FALSE;
   END_IF;
END_FUNCTION

ORGANIZATION_BLOCK "Main"   // OB1, LAD, ProgramCycle
TITLE = "Main Program Sweep (Cycle)"
{ S7_Optimized_Access := 'TRUE' }
VERSION : 0.1
   VAR_INPUT
      Initial_Call : Bool;   // Initial call of this OB
      Remanence : Bool;   // =True, if remanent data are available
   END_VAR
BEGIN

REGION Network 1
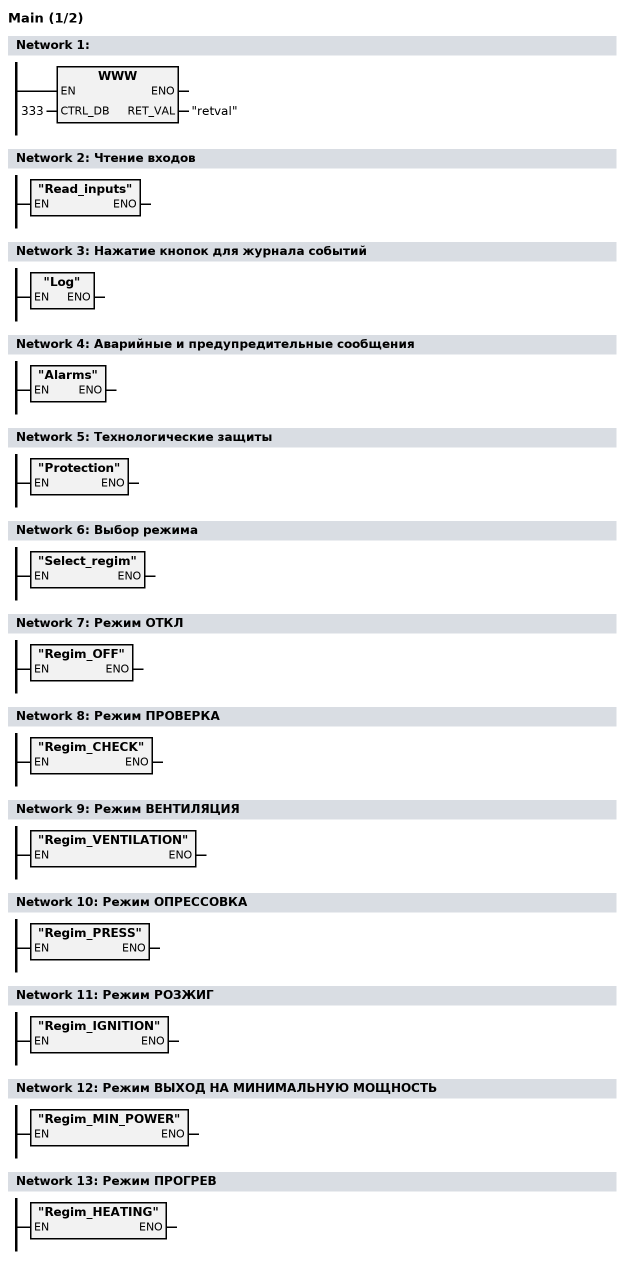
   "retval" := WWW(CTRL_DB := 333);
END_REGION

REGION Network 2: Чтение входов
   RUNG wire#powerrail
      "Read_inputs"()
   END_RUNG
   // the same network as SCL:
   "Read_inputs"();
END_REGION

REGION Network 3: Нажатие кнопок для журнала событий
   RUNG wire#powerrail
      "Log"()
   END_RUNG
   // the same network as SCL:
   "Log"();
END_REGION

REGION Network 4: Аварийные и предупредительные сообщения
   RUNG wire#powerrail
      "Alarms"()
   END_RUNG
   // the same network as SCL:
   "Alarms"();
END_REGION

REGION Network 5: Технологические защиты
   RUNG wire#powerrail
      "Protection"()
   END_RUNG
   // the same network as SCL:
   "Protection"();
END_REGION

REGION Network 6: Выбор режима
   RUNG wire#powerrail
      "Select_regim"()
   END_RUNG
   // the same network as SCL:
   "Select_regim"();
END_REGION

REGION Network 7: Режим ОТКЛ
   RUNG wire#powerrail
      "Regim_OFF"()
   END_RUNG
   // the same network as SCL:
   "Regim_OFF"();
END_REGION

REGION Network 8: Режим ПРОВЕРКА
   RUNG wire#powerrail
      "Regim_CHECK"()
   END_RUNG
   // the same network as SCL:
   "Regim_CHECK"();
END_REGION

REGION Network 9: Режим ВЕНТИЛЯЦИЯ
   RUNG wire#powerrail
      "Regim_VENTILATION"()
   END_RUNG
   // the same network as SCL:
   "Regim_VENTILATION"();
END_REGION

REGION Network 10: Режим ОПРЕССОВКА
   RUNG wire#powerrail
      "Regim_PRESS"()
   END_RUNG
   // the same network as SCL:
   "Regim_PRESS"();
END_REGION

REGION Network 11: Режим РОЗЖИГ
   RUNG wire#powerrail
      "Regim_IGNITION"()
   END_RUNG
   // the same network as SCL:
   "Regim_IGNITION"();
END_REGION

REGION Network 12: Режим ВЫХОД НА МИНИМАЛЬНУЮ МОЩНОСТЬ
   RUNG wire#powerrail
      "Regim_MIN_POWER"()
   END_RUNG
   // the same network as SCL:
   "Regim_MIN_POWER"();
END_REGION

REGION Network 13: Режим ПРОГРЕВ
   RUNG wire#powerrail
      "Regim_HEATING"()
   END_RUNG
   // the same network as SCL:
   "Regim_HEATING"();
END_REGION

REGION Network 14: Режим РАБОТА
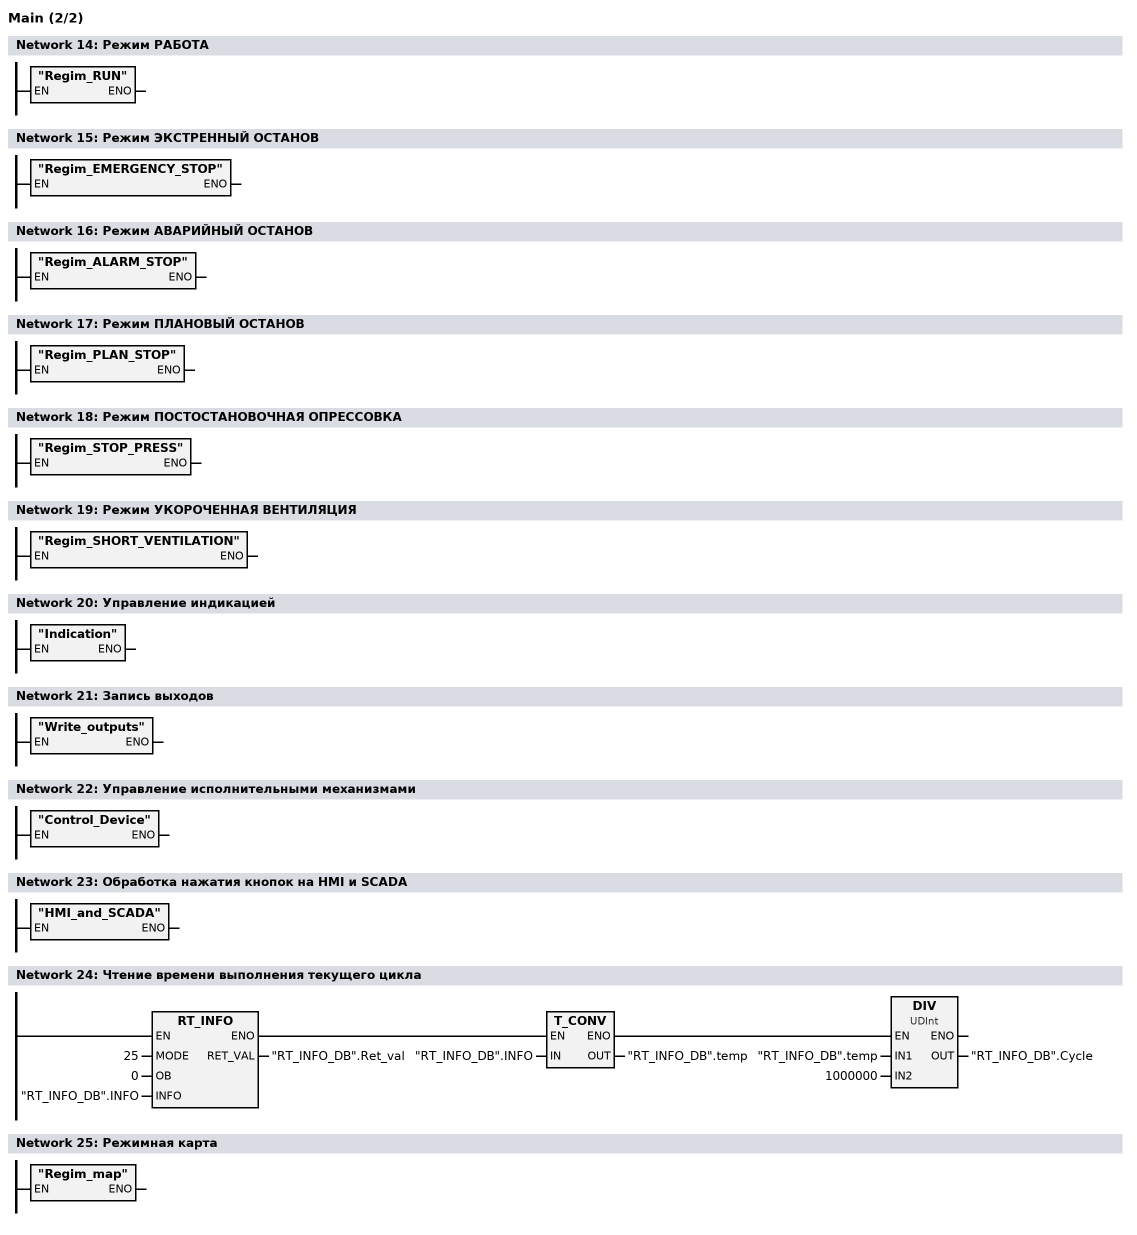
   RUNG wire#powerrail
      "Regim_RUN"()
   END_RUNG
   // the same network as SCL:
   "Regim_RUN"();
END_REGION

REGION Network 15: Режим ЭКСТРЕННЫЙ ОСТАНОВ
   RUNG wire#powerrail
      "Regim_EMERGENCY_STOP"()
   END_RUNG
   // the same network as SCL:
   "Regim_EMERGENCY_STOP"();
END_REGION

REGION Network 16: Режим АВАРИЙНЫЙ ОСТАНОВ
   RUNG wire#powerrail
      "Regim_ALARM_STOP"()
   END_RUNG
   // the same network as SCL:
   "Regim_ALARM_STOP"();
END_REGION

REGION Network 17: Режим ПЛАНОВЫЙ ОСТАНОВ
   RUNG wire#powerrail
      "Regim_PLAN_STOP"()
   END_RUNG
   // the same network as SCL:
   "Regim_PLAN_STOP"();
END_REGION

REGION Network 18: Режим ПОСТОСТАНОВОЧНАЯ ОПРЕССОВКА
   RUNG wire#powerrail
      "Regim_STOP_PRESS"()
   END_RUNG
   // the same network as SCL:
   "Regim_STOP_PRESS"();
END_REGION

REGION Network 19: Режим УКОРОЧЕННАЯ ВЕНТИЛЯЦИЯ
   RUNG wire#powerrail
      "Regim_SHORT_VENTILATION"()
   END_RUNG
   // the same network as SCL:
   "Regim_SHORT_VENTILATION"();
END_REGION

REGION Network 20: Управление индикацией
   RUNG wire#powerrail
      "Indication"()
   END_RUNG
   // the same network as SCL:
   "Indication"();
END_REGION

REGION Network 21: Запись выходов
   RUNG wire#powerrail
      "Write_outputs"()
   END_RUNG
   // the same network as SCL:
   "Write_outputs"();
END_REGION

REGION Network 22: Управление исполнительными механизмами
   RUNG wire#powerrail
      "Control_Device"()
   END_RUNG
   // the same network as SCL:
   "Control_Device"();
END_REGION

REGION Network 23: Обработка нажатия кнопок на HMI и SCADA
   RUNG wire#powerrail
      "HMI_and_SCADA"()
   END_RUNG
   // the same network as SCL:
   "HMI_and_SCADA"();
END_REGION

REGION Network 24: Чтение времени выполнения текущего цикла
   // ENO of a box is taken as its EN; it also drops when the box reports an error
   "RT_INFO_DB".Ret_val := RT_INFO(MODE := 25, OB := 0, INFO := "RT_INFO_DB".INFO);
   "RT_INFO_DB".temp := T_CONV(IN := "RT_INFO_DB".INFO);
   "RT_INFO_DB".Cycle := "RT_INFO_DB".temp / 1000000;
END_REGION

REGION Network 25: Режимная карта
   RUNG wire#powerrail
      "Regim_map"()
   END_RUNG
   // the same network as SCL:
   "Regim_map"();
END_REGION
END_ORGANIZATION_BLOCK

// folder: Regims

FUNCTION "Regim_OFF" : Void   // FC10, SCL
{ S7_Optimized_Access := 'TRUE' }
VERSION : 0.1
BEGIN
   (*Режим ОТКЛ*)
   (*таймеры*)
   (*процесс*)
   IF "Technology".Regim = 1 THEN
       CASE "Technology".Regim_off_step OF
           0:  // перевод управления всеми исполнительными устройствами в ручной режим
               "Control_ZRG".Mode:=FALSE;                  //ЗРГ
               "Control_ZRG".Mode_from_PLC := TRUE;
               "Control_ZDG".Mode:=FALSE;                  //ЗДГ
               "Control_ZDG".Avto_close := FALSE;
               "Control_ZDG".Avto_open := FALSE;
               "Control_ZDG".Avto_stop := FALSE;
               "Control_KB".Mode:=FALSE;                   //КБ
               "Control_KB".Avto_close := FALSE;
               "Control_KO".Mode:=FALSE;                   //КО
               "Control_KO".Avto_open := FALSE;
               "Control_KZ".Mode:=FALSE;                   //КЗ
               "Control_KZ".Avto_open := FALSE;
               "Control_PZK1".Mode:=FALSE;                 //ПЗК1
               "Control_PZK1".Avto_open := FALSE;
               "Control_PZK2".Mode:=FALSE;                 //ПЗК2
               "Control_PZK2".Avto_open := FALSE;
               "Control_IVN".Mode:=FALSE;                  //ИВН
               "Control_IVN".Avto_on := FALSE;
               "Control_ZDSV_before_boiler".Mode:=FALSE;   //ЗДСВ перед котлом
               "Control_ZDSV_before_boiler".Avto_close := FALSE;
               "Control_ZDSV_before_boiler".Avto_open := FALSE;
               "Control_ZDSV_before_boiler".Avto_stop := FALSE;
               "Control_ZDSV_after_boiler".Mode := FALSE;  //ЗДСВ после котла
               "Control_ZDSV_after_boiler".Avto_close := FALSE;
               "Control_ZDSV_after_boiler".Avto_open := FALSE;
               "Control_ZDSV_after_boiler".Avto_stop := FALSE;
               "Control_NAV".Mode:= FALSE;                 //НАВ
               "Control_NAV".Mode_from_PLC := TRUE;
               "Control_NAV".SP_PID := "RegMap".P_air_regim_map;
               "Control_NAV".Manual_close_from_PLC := FALSE;
               "Control_NAV".Manual_open_from_PLC := FALSE;
               "Control_NAD".Mode:= FALSE;                 //НАД
               "Control_NAD".Mode_from_PLC := TRUE;
               "Control_NAD".SP_PID := "RegMap".dP_furnace_regim_map;
               "Control_NAD".Manual_close_from_PLC := FALSE;
               "Control_NAD".Manual_open_from_PLC := FALSE;
               "Control_DV".Mode:= FALSE;                  //ДВ
               "Control_DV".Mode_from_PLC := TRUE;
               "Control_DV".SP_PID := "RegMap".P_air_regim_map;
               "Control_DV".Avto_Start := FALSE;
               "Control_DV".Avto_Stop := FALSE;
               "Control_DS".Mode:= FALSE;                  //ДС
               "Control_DS".Mode_from_PLC := TRUE;
               "Control_DS".SP_PID := "RegMap".dP_furnace_regim_map;
               "Control_DS".Avto_Start := FALSE;
               "Control_DS".Avto_Stop := FALSE;

           1:   //Ничего не делаем
               ;

           2:  //перевод всех клапанов в исходное состояние
               //все газовые клапана переводим в исходное состояние
               "Control_PZK1".Mode := TRUE;    //закрываем ПЗК1
               "Control_PZK1".Avto_open := FALSE;
               "Control_PZK2".Mode := TRUE;    //закрываем ПЗК2
               "Control_PZK2".Avto_open := FALSE;
               "Control_KO".Mode := TRUE;  //закрываем КО
               "Control_KO".Avto_open := FALSE;
               "Control_KZ".Mode := TRUE;  //закрываем КЗ
               "Control_KZ".Avto_open := FALSE;
               "Control_KB".Mode := TRUE;  //открываем КБ
               "Control_KB".Avto_close := FALSE;
               "Control_IVN".Mode := TRUE; //отключаем ИВН
               "Control_IVN".Avto_on := FALSE;

               "Control_ZRG".Mode := FALSE;                  //ЗРГ
               "Control_ZRG".Mode_from_PLC := TRUE;

               //контроль положения клапанов
               IF NOT "Sensors".PZK1_open.Value AND
                   NOT "Sensors".PZK2_not_close.Value AND
                   NOT "Sensors".KO_open.Value AND
                   NOT "Sensors".KZ_open.Value AND
                   NOT "Sensors".KB_close.Value THEN
                   "Technology".Regim_off_step := 3;
               END_IF;

           3:  //снимаем защиту Отключение ДВ
               "Alarms_and_warnings".Enable_Alarm_DV_off := FALSE;
               //отключение ДВ
               "Control_DV".Mode := TRUE;
               "Control_DV".Mode_from_PLC := FALSE;
               "Control_DV".Avto_Stop := TRUE;
               IF NOT "Sensors".DV_invertor_on.Value AND NOT "Sensors".DV_powergrid_on.Value THEN
                   //переход на следующий шаг
                   "Technology".Regim_off_step := 4;
               END_IF;

           4: //снимаем защиту Отключение ДС
               "Alarms_and_warnings".Enable_Alarm_DS_off := FALSE;
               //отключение ДС
               "Control_DS".Mode := TRUE;
               "Control_DS".Mode_from_PLC := FALSE;
               "Control_DS".Avto_Stop := TRUE;
               IF NOT "Sensors".DS_invertor_on.Value AND NOT "Sensors".DS_powergrid_on.Value THEN
                   "Technology".Regim_off_step := 0;
               END_IF;
           ELSE
               "Technology".Regim_off_step := 0;
       END_CASE;

       //нажатие кнопки ПЛАНОВЫЙ ОСТАНОВ
       IF "FRONT_Btn_Normal_stop_HMI" OR
           "FRONT_Btn_Normal_stop_SCADA" OR
           "FRONT_Btn_Alarm_stop_HMI" OR
           "FRONT_Btn_Alarm_stop_SCADA" THEN
           "Technology".Regim_off_step := 2;
       END_IF;
       //нажатие кнопки ВЕНТИЛЯЦИЯ
       IF "Sensors".Btn_Ventilation.Value OR
           "FRONT_Btn_Ventilation_HMI" OR
           "FRONT_Btn_Ventilation_SCADA" THEN
           "Message".OFF_Waiting_btn_ventilation := FALSE;
           "Technology".Regim := 3;    //переход на вентиляцию
           "Message".VENTILATION_not_initial_state_air := FALSE;
           "Message".VENTILATION_NAV_not_close := FALSE;
       ELSE
           "Message".OFF_Waiting_btn_ventilation := TRUE;
       END_IF;

   ELSE
       //Сброс текущего шага
       "Technology".Regim_off_step := 0;
       //Сброс всех сообщений по данному режиму
       "Message".OFF_Waiting_btn_ventilation := FALSE;
       "Message".OFF_Param_ventilation_not_norm := FALSE;
       //сброс таймеров
   END_IF;
END_FUNCTION

FUNCTION "Regim_CHECK" : Void   // FC12, SCL
{ S7_Optimized_Access := 'TRUE' }
VERSION : 0.1
BEGIN
   (*Режим ПРОВЕРКА*)
   (*таймеры*)
   (*процесс*)
   IF "Technology".Regim = 2 THEN
       ;
   ELSE
       "Technology".Regim_check_step := 0;
   END_IF;
END_FUNCTION

